LIN {X 0.323,Y -662.972,Z 876.335,A 0.000,B 0.000,C 90.000,E1 276.315} C_DIS
LIN {X 0.019,Y -659.761,Z 876.333,A 0.000,B 0.000,C 90.000,E1 275.853} C_DIS
LIN {X 0.348,Y -656.166,Z 876.330,A 0.000,B 0.000,C 90.000,E1 275.334} C_DIS
LIN {X -0.108,Y -650.680,Z 876.326,A 0.000,B 0.000,C 90.000,E1 274.759} C_DIS
LIN {X 0.134,Y -645.885,Z 876.324,A 0.000,B 0.000,C 90.000,E1 274.245} C_DIS
LIN {X -0.098,Y -638.071,Z 876.320,A 0.000,B 0.000,C 90.000,E1 273.555} C_DIS
LIN {X -0.003,Y -631.178,Z 876.317,A 0.000,B 0.000,C 90.000,E1 272.980} C_DIS
LIN {X -0.164,Y -623.612,Z 876.314,A 0.000,B 0.000,C 90.000,E1 272.465} C_DIS
LIN {X -0.009,Y -617.393,Z 876.312,A 0.000,B 0.000,C 90.000,E1 272.064} C_DIS
LIN {X -0.140,Y -610.911,Z 876.310,A 0.000,B 0.000,C 90.000,E1 271.718} C_DIS
LIN {X 0.108,Y -604.182,Z 876.308,A 0.000,B 0.000,C 90.000,E1 271.375} C_DIS
LIN {X 0.063,Y -597.337,Z 876.306,A 0.000,B 0.000,C 90.000,E1 271.088} C_DIS
LIN {X -0.214,Y -590.091,Z 876.305,A 0.000,B 0.000,C 90.000,E1 270.859} C_DIS
LIN {X -0.149,Y -584.631,Z 876.304,A 0.000,B 0.000,C 90.000,E1 270.688} C_DIS
LIN {X 0.237,Y -576.605,Z 876.303,A 0.000,B 0.000,C 90.000,E1 270.458} C_DIS
LIN {X 0.221,Y -569.921,Z 876.302,A 0.000,B 0.000,C 90.000,E1 270.344} C_DIS
LIN {X 0.254,Y -564.625,Z 876.302,A 0.000,B 0.000,C 90.000,E1 270.286} C_DIS
LIN {X 0.107,Y -553.667,Z 876.301,A 0.000,B 0.000,C 90.000,E1 270.229} C_DIS
LIN {X -0.050,Y -552.373,Z 876.301,A 0.000,B 0.000,C 90.000,E1 270.229} C_DIS
LIN {X 0.018,Y -549.331,Z 876.301,A 0.000,B 0.000,C 90.000,E1 270.115} C_DIS
LIN {X -0.108,Y -547.301,Z 876.300,A 0.000,B 0.000,C 90.000,E1 269.943} C_DIS
LIN {X -0.153,Y -546.410,Z 876.298,A 0.000,B 0.000,C 90.000,E1 269.714} C_DIS
LIN {X 0.190,Y -545.549,Z 876.296,A 0.000,B 0.000,C 90.000,E1 269.255} C_DIS
LIN {X 0.218,Y -541.822,Z 876.272,A 0.000,B 0.000,C 90.000,E1 265.008} C_DIS
LIN {X -0.161,Y -541.097,Z 876.266,A 0.000,B 0.000,C 90.000,E1 263.913} C_DIS
LIN {X 0.056,Y -540.026,Z 876.258,A 0.000,B 0.000,C 90.000,E1 262.470} C_DIS
LIN {X 0.242,Y -538.664,Z 876.250,A 0.000,B 0.000,C 90.000,E1 261.027} C_DIS
LIN {X -0.117,Y -537.550,Z 876.244,A 0.000,B 0.000,C 90.000,E1 259.926} C_DIS
LIN {X -0.273,Y -535.768,Z 876.234,A 0.000,B 0.000,C 90.000,E1 258.229} C_DIS
LIN {X -0.051,Y -534.476,Z 876.228,A 0.000,B 0.000,C 90.000,E1 257.061} C_DIS
LIN {X -0.248,Y -533.064,Z 876.222,A 0.000,B 0.000,C 90.000,E1 255.936} C_DIS
LIN {X -0.214,Y -530.574,Z 876.211,A 0.000,B 0.000,C 90.000,E1 253.921} C_DIS
LIN {X 0.057,Y -528.202,Z 876.199,A 0.000,B 0.000,C 90.000,E1 251.873} C_DIS
LIN {X -0.252,Y -527.077,Z 876.195,A 0.000,B 0.000,C 90.000,E1 251.040} C_DIS
LIN {X -0.063,Y -525.191,Z 876.187,A 0.000,B 0.000,C 90.000,E1 249.571} C_DIS
LIN {X -0.073,Y -523.643,Z 876.180,A 0.000,B 0.000,C 90.000,E1 248.411} C_DIS
LIN {X 0.243,Y -521.461,Z 876.172,A 0.000,B 0.000,C 90.000,E1 246.922} C_DIS
LIN {X -0.107,Y -519.733,Z 876.166,A 0.000,B 0.000,C 90.000,E1 245.793} C_DIS
LIN {X -0.123,Y -517.477,Z 876.157,A 0.000,B 0.000,C 90.000,E1 244.332} C_DIS
LIN {X 0.157,Y -515.575,Z 876.151,A 0.000,B 0.000,C 90.000,E1 243.127} C_DIS
LIN {X -0.056,Y -512.523,Z 876.141,A 0.000,B 0.000,C 90.000,E1 241.385} C_DIS
LIN {X -0.098,Y -509.431,Z 876.131,A 0.000,B 0.000,C 90.000,E1 239.616} C_DIS
LIN {X 0.092,Y -507.327,Z 876.125,A 0.000,B 0.000,C 90.000,E1 238.408} C_DIS
LIN {X 0.136,Y -504.494,Z 876.116,A 0.000,B 0.000,C 90.000,E1 236.914} C_DIS
LIN {X 0.107,Y -502.069,Z 876.110,A 0.000,B 0.000,C 90.000,E1 235.722} C_DIS
LIN {X 0.288,Y -500.765,Z 876.106,A 0.000,B 0.000,C 90.000,E1 235.102} C_DIS
LIN {X 0.079,Y -497.210,Z 876.098,A 0.000,B 0.000,C 90.000,E1 233.623} C_DIS
LIN {X -0.042,Y -492.982,Z 876.088,A 0.000,B 0.000,C 90.000,E1 231.823} C_DIS
LIN {X 0.202,Y -489.383,Z 876.079,A 0.000,B 0.000,C 90.000,E1 230.275} C_DIS
LIN {X -0.143,Y -486.645,Z 876.073,A 0.000,B 0.000,C 90.000,E1 229.094} C_DIS
LIN {X 0.110,Y -483.868,Z 876.066,A 0.000,B 0.000,C 90.000,E1 227.838} C_DIS
LIN {X 0.253,Y -479.873,Z 876.056,A 0.000,B 0.000,C 90.000,E1 225.972} C_DIS
LIN {X 0.285,Y -475.776,Z 876.045,A 0.000,B 0.000,C 90.000,E1 224.109} C_DIS
LIN {X -0.199,Y -472.305,Z 876.037,A 0.000,B 0.000,C 90.000,E1 222.609} C_DIS
LIN {X 0.100,Y -467.450,Z 876.024,A 0.000,B 0.000,C 90.000,E1 220.378} C_DIS
LIN {X 0.020,Y -462.719,Z 876.012,A 0.000,B 0.000,C 90.000,E1 218.177} C_DIS
LIN {X -0.203,Y -458.741,Z 876.002,A 0.000,B 0.000,C 90.000,E1 216.297} C_DIS
LIN {X 0.215,Y -454.685,Z 875.991,A 0.000,B 0.000,C 90.000,E1 214.326} C_DIS
LIN {X 0.130,Y -452.624,Z 875.986,A 0.000,B 0.000,C 90.000,E1 213.372} C_DIS
LIN {X -0.102,Y -448.540,Z 875.975,A 0.000,B 0.000,C 90.000,E1 211.465} C_DIS
LIN {X -0.219,Y -443.633,Z 875.962,A 0.000,B 0.000,C 90.000,E1 209.205} C_DIS
LIN {X 0.212,Y -440.087,Z 875.953,A 0.000,B 0.000,C 90.000,E1 207.513} C_DIS
LIN {X 0.215,Y -435.105,Z 875.940,A 0.000,B 0.000,C 90.000,E1 205.207} C_DIS
LIN {X -0.102,Y -430.943,Z 875.929,A 0.000,B 0.000,C 90.000,E1 203.259} C_DIS
LIN {X -0.085,Y -426.161,Z 875.916,A 0.000,B 0.000,C 90.000,E1 200.918} C_DIS
LIN {X 0.085,Y -422.719,Z 875.907,A 0.000,B 0.000,C 90.000,E1 199.214} C_DIS
LIN {X 0.177,Y -419.410,Z 875.897,A 0.000,B 0.000,C 90.000,E1 197.511} C_DIS
LIN {X -0.207,Y -416.674,Z 875.890,A 0.000,B 0.000,C 90.000,E1 196.205} C_DIS
LIN {X -0.081,Y -413.195,Z 875.880,A 0.000,B 0.000,C 90.000,E1 194.481} C_DIS
LIN {X 0.010,Y -408.527,Z 875.867,A 0.000,B 0.000,C 90.000,E1 192.063} C_DIS
LIN {X 0.161,Y -405.858,Z 875.859,A 0.000,B 0.000,C 90.000,E1 190.658} C_DIS
LIN {X 0.195,Y -402.402,Z 875.850,A 0.000,B 0.000,C 90.000,E1 188.916} C_DIS
LIN {X 0.064,Y -397.475,Z 875.836,A 0.000,B 0.000,C 90.000,E1 186.486} C_DIS
LIN {X 0.194,Y -390.868,Z 875.815,A 0.000,B 0.000,C 90.000,E1 182.579} C_DIS
LIN {X 0.078,Y -387.709,Z 875.803,A 0.000,B 0.000,C 90.000,E1 180.458} C_DIS
LIN {X 0.084,Y -385.689,Z 875.795,A 0.000,B 0.000,C 90.000,E1 179.026} C_DIS
LIN {X -0.046,Y -382.997,Z 875.785,A 0.000,B 0.000,C 90.000,E1 177.249} C_DIS
LIN {X -0.087,Y -380.876,Z 875.777,A 0.000,B 0.000,C 90.000,E1 175.812} C_DIS
LIN {X -0.123,Y -377.307,Z 875.763,A 0.000,B 0.000,C 90.000,E1 173.280} C_DIS
LIN {X 0.154,Y -375.585,Z 875.755,A 0.000,B 0.000,C 90.000,E1 171.781} C_DIS
LIN {X 0.082,Y -374.388,Z 875.746,A 0.000,B 0.000,C 90.000,E1 170.330} C_DIS
LIN {X 0.175,Y -373.752,Z 875.740,A 0.000,B 0.000,C 90.000,E1 169.218} C_DIS
LIN {X -0.176,Y -373.799,Z 875.734,A 0.000,B 0.000,C 90.000,E1 168.173} C_DIS
LIN {X 0.030,Y -374.075,Z 875.730,A 0.000,B 0.000,C 90.000,E1 167.409} C_DIS
LIN {X -0.125,Y -374.536,Z 875.726,A 0.000,B 0.000,C 90.000,E1 166.700} C_DIS
LIN {X 0.103,Y -375.301,Z 875.723,A 0.000,B 0.000,C 90.000,E1 166.117} C_DIS
LIN {X 0.082,Y -376.304,Z 875.721,A 0.000,B 0.000,C 90.000,E1 165.700} C_DIS
LIN {X 0.058,Y -377.044,Z 875.719,A 0.000,B 0.000,C 90.000,E1 165.338} C_DIS
LIN {X -0.058,Y -378.009,Z 875.717,A 0.000,B 0.000,C 90.000,E1 164.991} C_DIS
LIN {X 0.036,Y -379.120,Z 875.715,A 0.000,B 0.000,C 90.000,E1 164.629} C_DIS
LIN {X -0.079,Y -382.383,Z 875.712,A 0.000,B 0.000,C 90.000,E1 164.102} C_DIS
LIN {X -0.081,Y -383.396,Z 875.711,A 0.000,B 0.000,C 90.000,E1 163.921} C_DIS
LIN {X -0.077,Y -384.658,Z 875.710,A 0.000,B 0.000,C 90.000,E1 163.740} C_DIS
LIN {X 0.042,Y -390.123,Z 875.707,A 0.000,B 0.000,C 90.000,E1 163.196} C_DIS
LIN {X -0.218,Y -392.050,Z 875.706,A 0.000,B 0.000,C 90.000,E1 163.087} C_DIS
LIN {X -0.034,Y -398.644,Z 875.704,A 0.000,B 0.000,C 90.000,E1 162.670} C_DIS
LIN {X -0.002,Y -417.692,Z 875.698,A 0.000,B 0.000,C 90.000,E1 161.692} C_DIS
LIN {X 0.178,Y -422.461,Z 875.697,A 0.000,B 0.000,C 90.000,E1 161.402} C_DIS
LIN {X -0.122,Y -428.928,Z 875.695,A 0.000,B 0.000,C 90.000,E1 161.040} C_DIS
LIN {X -0.202,Y -438.322,Z 875.691,A 0.000,B 0.000,C 90.000,E1 160.369} C_DIS
LIN {X -0.136,Y -446.051,Z 875.687,A 0.000,B 0.000,C 90.000,E1 159.752} C_DIS
LIN {X -0.042,Y -456.665,Z 875.682,A 0.000,B 0.000,C 90.000,E1 158.847} C_DIS
LIN {X -0.125,Y -459.495,Z 875.681,A 0.000,B 0.000,C 90.000,E1 158.592} C_DIS
LIN {X -0.089,Y -469.554,Z 875.675,A 0.000,B 0.000,C 90.000,E1 157.592} C_DIS
LIN {X 0.090,Y -479.076,Z 875.670,A 0.000,B 0.000,C 90.000,E1 156.538} C_DIS
LIN {X -0.175,Y -489.344,Z 875.663,A 0.000,B 0.000,C 90.000,E1 155.357} C_DIS
LIN {X 0.120,Y -496.471,Z 875.658,A 0.000,B 0.000,C 90.000,E1 154.409} C_DIS
LIN {X -0.141,Y -504.231,Z 875.652,A 0.000,B 0.000,C 90.000,E1 153.384} C_DIS
LIN {X 0.054,Y -509.663,Z 875.648,A 0.000,B 0.000,C 90.000,E1 152.615} C_DIS
LIN {X 0.145,Y -519.842,Z 875.640,A 0.000,B 0.000,C 90.000,E1 151.129} C_DIS
LIN {X 0.128,Y -525.696,Z 875.635,A 0.000,B 0.000,C 90.000,E1 150.255} C_DIS
LIN {X -0.087,Y -531.123,Z 875.630,A 0.000,B 0.000,C 90.000,E1 149.410} C_DIS
LIN {X 0.024,Y -536.329,Z 875.625,A 0.000,B 0.000,C 90.000,E1 148.535} C_DIS
LIN {X -0.268,Y -539.600,Z 875.622,A 0.000,B 0.000,C 90.000,E1 147.995} C_DIS
LIN {X -0.137,Y -548.333,Z 875.613,A 0.000,B 0.000,C 90.000,E1 146.421} C_DIS
LIN {X 0.345,Y -553.510,Z 875.608,A 0.000,B 0.000,C 90.000,E1 145.388} C_DIS
LIN {X -0.216,Y -557.743,Z 875.603,A 0.000,B 0.000,C 90.000,E1 144.609} C_DIS
LIN {X -0.165,Y -561.241,Z 875.599,A 0.000,B 0.000,C 90.000,E1 143.909} C_DIS
LIN {X 0.135,Y -567.608,Z 875.593,A 0.000,B 0.000,C 90.000,E1 142.637} C_DIS
LIN {X -0.083,Y -576.334,Z 875.583,A 0.000,B 0.000,C 90.000,E1 140.884} C_DIS
LIN {X 0.091,Y -581.515,Z 875.577,A 0.000,B 0.000,C 90.000,E1 139.784} C_DIS
LIN {X 0.276,Y -586.418,Z 875.571,A 0.000,B 0.000,C 90.000,E1 138.690} C_DIS
LIN {X -0.131,Y -595.235,Z 875.560,A 0.000,B 0.000,C 90.000,E1 136.863} C_DIS
LIN {X 0.038,Y -601.513,Z 875.553,A 0.000,B 0.000,C 90.000,E1 135.526} C_DIS
LIN {X -0.276,Y -603.439,Z 875.551,A 0.000,B 0.000,C 90.000,E1 135.162} C_DIS
LIN {X 0.041,Y -609.364,Z 875.544,A 0.000,B 0.000,C 90.000,E1 133.824} C_DIS
LIN {X 0.187,Y -614.049,Z 875.538,A 0.000,B 0.000,C 90.000,E1 132.771} C_DIS
LIN {X -0.191,Y -619.680,Z 875.531,A 0.000,B 0.000,C 90.000,E1 131.515} C_DIS
LIN {X 0.128,Y -624.020,Z 875.525,A 0.000,B 0.000,C 90.000,E1 130.458} C_DIS
LIN {X 0.110,Y -628.089,Z 875.519,A 0.000,B 0.000,C 90.000,E1 129.439} C_DIS
LIN {X 0.024,Y -632.995,Z 875.512,A 0.000,B 0.000,C 90.000,E1 128.177} C_DIS
LIN {X 0.131,Y -636.916,Z 875.507,A 0.000,B 0.000,C 90.000,E1 127.156} C_DIS
LIN {X -0.093,Y -640.736,Z 875.501,A 0.000,B 0.000,C 90.000,E1 126.171} C_DIS
LIN {X 0.223,Y -643.496,Z 875.497,A 0.000,B 0.000,C 90.000,E1 125.391} C_DIS
LIN {X -0.393,Y -647.581,Z 875.490,A 0.000,B 0.000,C 90.000,E1 124.199} C_DIS
LIN {X 0.056,Y -650.606,Z 875.484,A 0.000,B 0.000,C 90.000,E1 123.166} C_DIS
LIN {X -0.356,Y -653.285,Z 875.479,A 0.000,B 0.000,C 90.000,E1 122.212} C_DIS
LIN {X -0.281,Y -655.064,Z 875.475,A 0.000,B 0.000,C 90.000,E1 121.465} C_DIS
LIN {X 0.031,Y -657.619,Z 875.468,A 0.000,B 0.000,C 90.000,E1 120.207} C_DIS
LIN {X 0.262,Y -659.283,Z 875.462,A 0.000,B 0.000,C 90.000,E1 119.205} C_DIS
LIN {X 0.063,Y -660.434,Z 875.458,A 0.000,B 0.000,C 90.000,E1 118.487} C_DIS
LIN {X 0.006,Y -661.948,Z 875.453,A 0.000,B 0.000,C 90.000,E1 117.513} C_DIS
LIN {X -0.173,Y -663.047,Z 875.449,A 0.000,B 0.000,C 90.000,E1 116.796} C_DIS
LIN {X 0.101,Y -664.310,Z 875.443,A 0.000,B 0.000,C 90.000,E1 115.796} C_DIS
LIN {X 0.082,Y -665.051,Z 875.438,A 0.000,B 0.000,C 90.000,E1 114.823} C_DIS
LIN {X 0.097,Y -665.286,Z 875.435,A 0.000,B 0.000,C 90.000,E1 114.335} C_DIS
LIN {X 0.389,Y -665.304,Z 875.433,A 0.000,B 0.000,C 90.000,E1 113.823} C_DIS
LIN {X -0.196,Y -664.753,Z 875.430,A 0.000,B 0.000,C 90.000,E1 113.387} C_DIS
LIN {X -0.054,Y -664.380,Z 875.429,A 0.000,B 0.000,C 90.000,E1 113.131} C_DIS
LIN {X 0.035,Y -661.702,Z 875.425,A 0.000,B 0.000,C 90.000,E1 112.514} C_DIS
LIN {X 0.102,Y -660.802,Z 875.424,A 0.000,B 0.000,C 90.000,E1 112.386} C_DIS
LIN {X -0.021,Y -658.470,Z 875.423,A 0.000,B 0.000,C 90.000,E1 112.153} C_DIS
LIN {X 0.044,Y -657.015,Z 875.422,A 0.000,B 0.000,C 90.000,E1 111.972} C_DIS
LIN {X 0.102,Y -655.691,Z 875.421,A 0.000,B 0.000,C 90.000,E1 111.844} C_DIS
LIN {X -0.054,Y -652.134,Z 875.420,A 0.000,B 0.000,C 90.000,E1 111.642} C_DIS
LIN {X -0.203,Y -647.809,Z 875.419,A 0.000,B 0.000,C 90.000,E1 111.408} C_DIS
LIN {X -0.086,Y -641.358,Z 875.418,A 0.000,B 0.000,C 90.000,E1 111.153} C_DIS
LIN {X 0.165,Y -630.848,Z 875.416,A 0.000,B 0.000,C 90.000,E1 110.791} C_DIS
LIN {X -0.177,Y -625.740,Z 875.415,A 0.000,B 0.000,C 90.000,E1 110.663} C_DIS
LIN {X 0.152,Y -621.263,Z 875.414,A 0.000,B 0.000,C 90.000,E1 110.482} C_DIS
LIN {X 0.066,Y -619.301,Z 875.414,A 0.000,B 0.000,C 90.000,E1 110.429} C_DIS
LIN {X -0.245,Y -610.433,Z 875.412,A 0.000,B 0.000,C 90.000,E1 110.120} C_DIS
LIN {X 0.043,Y -601.778,Z 875.410,A 0.000,B 0.000,C 90.000,E1 109.704} C_DIS
LIN {X -0.266,Y -591.984,Z 875.407,A 0.000,B 0.000,C 90.000,E1 109.268} C_DIS
LIN {X -0.114,Y -587.313,Z 875.406,A 0.000,B 0.000,C 90.000,E1 109.033} C_DIS
LIN {X -0.312,Y -578.780,Z 875.404,A 0.000,B 0.000,C 90.000,E1 108.725} C_DIS
LIN {X -0.196,Y -565.827,Z 875.402,A 0.000,B 0.000,C 90.000,E1 108.308} C_DIS
LIN {X 0.212,Y -562.764,Z 875.401,A 0.000,B 0.000,C 90.000,E1 108.127} C_DIS
LIN {X 0.156,Y -561.424,Z 875.400,A 0.000,B 0.000,C 90.000,E1 108.055} C_DIS
LIN {X -0.142,Y -559.895,Z 875.400,A 0.000,B 0.000,C 90.000,E1 107.946} C_DIS
LIN {X 0.091,Y -558.501,Z 875.398,A 0.000,B 0.000,C 90.000,E1 107.583} C_DIS
LIN {X 0.253,Y -558.033,Z 875.396,A 0.000,B 0.000,C 90.000,E1 107.221} C_DIS
LIN {X 0.017,Y -557.954,Z 875.390,A 0.000,B 0.000,C 90.000,E1 106.134} C_DIS
LIN {X 0.186,Y -559.024,Z 875.373,A 0.000,B 0.000,C 90.000,E1 103.063} C_DIS
LIN {X -0.032,Y -560.051,Z 875.363,A 0.000,B 0.000,C 90.000,E1 101.422} C_DIS
LIN {X -0.030,Y -561.573,Z 875.351,A 0.000,B 0.000,C 90.000,E1 99.208} C_DIS
LIN {X 0.167,Y -562.701,Z 875.342,A 0.000,B 0.000,C 90.000,E1 97.530} C_DIS
LIN {X 0.232,Y -563.537,Z 875.334,A 0.000,B 0.000,C 90.000,E1 96.144} C_DIS
LIN {X 0.301,Y -564.171,Z 875.327,A 0.000,B 0.000,C 90.000,E1 94.759} C_DIS
LIN {X -0.276,Y -564.766,Z 875.319,A 0.000,B 0.000,C 90.000,E1 93.440} C_DIS
LIN {X -0.271,Y -565.203,Z 875.311,A 0.000,B 0.000,C 90.000,E1 92.064} C_DIS
LIN {X -0.260,Y -565.669,Z 875.304,A 0.000,B 0.000,C 90.000,E1 90.688} C_DIS
LIN {X -0.140,Y -566.011,Z 875.295,A 0.000,B 0.000,C 90.000,E1 89.026} C_DIS
LIN {X -0.117,Y -566.258,Z 875.287,A 0.000,B 0.000,C 90.000,E1 87.650} C_DIS
LIN {X 0.171,Y -566.628,Z 875.276,A 0.000,B 0.000,C 90.000,E1 85.698} C_DIS
LIN {X -0.216,Y -566.879,Z 875.267,A 0.000,B 0.000,C 90.000,E1 84.090} C_DIS
LIN {X 0.176,Y -567.282,Z 875.256,A 0.000,B 0.000,C 90.000,E1 82.129} C_DIS
LIN {X 0.189,Y -567.890,Z 875.246,A 0.000,B 0.000,C 90.000,E1 80.208} C_DIS
LIN {X -0.146,Y -568.783,Z 875.234,A 0.000,B 0.000,C 90.000,E1 78.049} C_DIS
LIN {X 0.029,Y -569.281,Z 875.227,A 0.000,B 0.000,C 90.000,E1 76.937} C_DIS
LIN {X 0.154,Y -569.891,Z 875.218,A 0.000,B 0.000,C 90.000,E1 75.283} C_DIS
LIN {X 0.104,Y -570.360,Z 875.211,A 0.000,B 0.000,C 90.000,E1 73.921} C_DIS
LIN {X 0.042,Y -570.629,Z 875.205,A 0.000,B 0.000,C 90.000,E1 72.834} C_DIS
LIN {X -0.212,Y -570.967,Z 875.196,A 0.000,B 0.000,C 90.000,E1 71.221} C_DIS
LIN {X 0.255,Y -571.157,Z 875.185,A 0.000,B 0.000,C 90.000,E1 69.263} C_DIS
LIN {X 0.195,Y -571.268,Z 875.174,A 0.000,B 0.000,C 90.000,E1 67.358} C_DIS
LIN {X 0.162,Y -571.241,Z 875.167,A 0.000,B 0.000,C 90.000,E1 65.997} C_DIS
LIN {X -0.163,Y -571.153,Z 875.159,A 0.000,B 0.000,C 90.000,E1 64.665} C_DIS
LIN {X 0.277,Y -571.005,Z 875.152,A 0.000,B 0.000,C 90.000,E1 63.256} C_DIS
LIN {X 0.209,Y -570.687,Z 875.144,A 0.000,B 0.000,C 90.000,E1 61.897} C_DIS
LIN {X 0.238,Y -570.133,Z 875.135,A 0.000,B 0.000,C 90.000,E1 60.255} C_DIS
LIN {X 0.001,Y -569.754,Z 875.130,A 0.000,B 0.000,C 90.000,E1 59.459} C_DIS
LIN {X 0.178,Y -568.873,Z 875.123,A 0.000,B 0.000,C 90.000,E1 58.074} C_DIS
LIN {X 0.224,Y -568.272,Z 875.118,A 0.000,B 0.000,C 90.000,E1 57.248} C_DIS
LIN {X 0.267,Y -567.521,Z 875.114,A 0.000,B 0.000,C 90.000,E1 56.421} C_DIS
LIN {X 0.303,Y -566.647,Z 875.109,A 0.000,B 0.000,C 90.000,E1 55.595} C_DIS
LIN {X -0.021,Y -565.339,Z 875.103,A 0.000,B 0.000,C 90.000,E1 54.529} C_DIS
LIN {X 0.098,Y -563.814,Z 875.097,A 0.000,B 0.000,C 90.000,E1 53.417} C_DIS
LIN {X 0.077,Y -562.076,Z 875.091,A 0.000,B 0.000,C 90.000,E1 52.316} C_DIS
LIN {X 0.030,Y -560.593,Z 875.086,A 0.000,B 0.000,C 90.000,E1 51.492} C_DIS
LIN {X -0.219,Y -559.517,Z 875.083,A 0.000,B 0.000,C 90.000,E1 50.964} C_DIS
LIN {X -0.030,Y -557.698,Z 875.078,A 0.000,B 0.000,C 90.000,E1 50.114} C_DIS
LIN {X -0.214,Y -555.497,Z 875.074,A 0.000,B 0.000,C 90.000,E1 49.299} C_DIS
LIN {X -0.058,Y -553.014,Z 875.069,A 0.000,B 0.000,C 90.000,E1 48.447} C_DIS
LIN {X 0.058,Y -551.206,Z 875.066,A 0.000,B 0.000,C 90.000,E1 47.877} C_DIS
LIN {X -0.203,Y -547.058,Z 875.060,A 0.000,B 0.000,C 90.000,E1 46.782} C_DIS
LIN {X -0.165,Y -544.823,Z 875.057,A 0.000,B 0.000,C 90.000,E1 46.215} C_DIS
LIN {X -0.338,Y -543.053,Z 875.054,A 0.000,B 0.000,C 90.000,E1 45.810} C_DIS
LIN {X -0.139,Y -539.772,Z 875.050,A 0.000,B 0.000,C 90.000,E1 45.081} C_DIS
LIN {X 0.027,Y -536.128,Z 875.046,A 0.000,B 0.000,C 90.000,E1 44.352} C_DIS
LIN {X -0.191,Y -533.846,Z 875.044,A 0.000,B 0.000,C 90.000,E1 43.947} C_DIS
LIN {X 0.083,Y -528.644,Z 875.039,A 0.000,B 0.000,C 90.000,E1 43.056} C_DIS
LIN {X 0.208,Y -525.927,Z 875.037,A 0.000,B 0.000,C 90.000,E1 42.609} C_DIS
LIN {X -0.114,Y -521.051,Z 875.033,A 0.000,B 0.000,C 90.000,E1 41.919} C_DIS
LIN {X -0.025,Y -517.968,Z 875.030,A 0.000,B 0.000,C 90.000,E1 41.472} C_DIS
LIN {X -0.283,Y -511.277,Z 875.026,A 0.000,B 0.000,C 90.000,E1 40.620} C_DIS
LIN {X -0.128,Y -506.473,Z 875.022,A 0.000,B 0.000,C 90.000,E1 40.011} C_DIS
LIN {X 0.003,Y -501.274,Z 875.019,A 0.000,B 0.000,C 90.000,E1 39.402} C_DIS
LIN {X 0.104,Y -494.460,Z 875.015,A 0.000,B 0.000,C 90.000,E1 38.669} C_DIS
LIN {X 0.002,Y -490.260,Z 875.013,A 0.000,B 0.000,C 90.000,E1 38.257} C_DIS
LIN {X 0.017,Y -483.079,Z 875.009,A 0.000,B 0.000,C 90.000,E1 37.569} C_DIS
LIN {X -0.046,Y -475.646,Z 875.005,A 0.000,B 0.000,C 90.000,E1 36.916} C_DIS
LIN {X -0.017,Y -465.064,Z 875.000,A 0.000,B 0.000,C 90.000,E1 36.011} C_DIS
LIN {X -0.104,Y -452.656,Z 874.995,A 0.000,B 0.000,C 90.000,E1 35.025} C_DIS
LIN {X -0.065,Y -443.282,Z 874.990,A 0.000,B 0.000,C 90.000,E1 34.278} C_DIS
LIN {X 0.069,Y -421.693,Z 874.981,A 0.000,B 0.000,C 90.000,E1 32.498} C_DIS
LIN {X 0.024,Y -406.598,Z 874.973,A 0.000,B 0.000,C 90.000,E1 31.131} C_DIS
LIN {X -0.032,Y -399.449,Z 874.969,A 0.000,B 0.000,C 90.000,E1 30.413} C_DIS
LIN {X -0.157,Y -394.956,Z 874.966,A 0.000,B 0.000,C 90.000,E1 29.873} C_DIS
LIN {X 0.010,Y -392.401,Z 874.963,A 0.000,B 0.000,C 90.000,E1 29.411} C_DIS
LIN {X -0.057,Y -391.569,Z 874.962,A 0.000,B 0.000,C 90.000,E1 29.155} C_DIS
LIN {X 0.062,Y -390.550,Z 874.961,A 0.000,B 0.000,C 90.000,E1 28.871} C_DIS
LIN {X -0.008,Y -389.735,Z 874.958,A 0.000,B 0.000,C 90.000,E1 28.437} C_DIS
LIN {X 0.180,Y -389.516,Z 874.957,A 0.000,B 0.000,C 90.000,E1 28.231} C_DIS
LIN {X -0.109,Y -389.463,Z 874.954,A 0.000,B 0.000,C 90.000,E1 27.719} C_DIS
LIN {X 0.081,Y -389.305,Z 874.952,A 0.000,B 0.000,C 90.000,E1 27.334} C_DIS
LIN {X -0.034,Y -389.940,Z 874.944,A 0.000,B 0.000,C 90.000,E1 25.924} C_DIS
LIN {X 0.082,Y -391.522,Z 874.932,A 0.000,B 0.000,C 90.000,E1 23.770} C_DIS
LIN {X 0.169,Y -394.134,Z 874.916,A 0.000,B 0.000,C 90.000,E1 20.918} C_DIS
LIN {X -0.081,Y -396.351,Z 874.905,A 0.000,B 0.000,C 90.000,E1 18.833} C_DIS
LIN {X -0.091,Y -399.250,Z 874.891,A 0.000,B 0.000,C 90.000,E1 16.370} C_DIS
LIN {X 0.149,Y -402.374,Z 874.877,A 0.000,B 0.000,C 90.000,E1 13.883} C_DIS
LIN {X -0.094,Y -405.837,Z 874.864,A 0.000,B 0.000,C 90.000,E1 11.478} C_DIS
LIN {X 0.064,Y -410.729,Z 874.846,A 0.000,B 0.000,C 90.000,E1 8.341} C_DIS
LIN {X -0.167,Y -415.542,Z 874.831,A 0.000,B 0.000,C 90.000,E1 5.625} C_DIS
LIN {X 0.079,Y -420.777,Z 874.816,A 0.000,B 0.000,C 90.000,E1 2.865} C_DIS
LIN {X -0.204,Y -428.386,Z 874.797,A 0.000,B 0.000,C 90.000,E1 359.484} C_DIS
LIN {X 0.000,Y -434.970,Z 874.782,A 0.000,B 0.000,C 90.000,E1 356.788} C_DIS
LIN {X -0.040,Y -438.339,Z 874.775,A 0.000,B 0.000,C 90.000,E1 355.469} C_DIS
LIN {X 0.144,Y -439.863,Z 874.772,A 0.000,B 0.000,C 90.000,E1 354.951} C_DIS
LIN {X -0.037,Y -442.283,Z 874.769,A 0.000,B 0.000,C 90.000,E1 354.375} C_DIS
LIN {X 0.016,Y -443.078,Z 874.768,A 0.000,B 0.000,C 90.000,E1 354.204} C_DIS
LIN {X -0.165,Y -445.091,Z 874.766,A 0.000,B 0.000,C 90.000,E1 353.913} C_DIS
LIN {X -0.003,Y -450.120,Z 874.764,A 0.000,B 0.000,C 90.000,E1 353.451} C_DIS
LIN {X -0.228,Y -455.758,Z 874.762,A 0.000,B 0.000,C 90.000,E1 353.166} C_DIS
LIN {X 0.240,Y -470.201,Z 874.758,A 0.000,B 0.000,C 90.000,E1 352.470} C_DIS
LIN {X -0.118,Y -473.472,Z 874.758,A 0.000,B 0.000,C 90.000,E1 352.356} C_DIS
LIN {X -0.073,Y -483.315,Z 874.755,A 0.000,B 0.000,C 90.000,E1 351.837} C_DIS
LIN {X 0.204,Y -492.976,Z 874.752,A 0.000,B 0.000,C 90.000,E1 351.254} C_DIS
LIN {X -0.252,Y -504.167,Z 874.748,A 0.000,B 0.000,C 90.000,E1 350.622} C_DIS
LIN {X -0.060,Y -512.046,Z 874.745,A 0.000,B 0.000,C 90.000,E1 350.095} C_DIS
LIN {X -0.012,Y -521.344,Z 874.741,A 0.000,B 0.000,C 90.000,E1 349.454} C_DIS
LIN {X -0.201,Y -528.953,Z 874.738,A 0.000,B 0.000,C 90.000,E1 348.926} C_DIS
LIN {X -0.130,Y -534.869,Z 874.736,A 0.000,B 0.000,C 90.000,E1 348.465} C_DIS
LIN {X 0.213,Y -542.002,Z 874.733,A 0.000,B 0.000,C 90.000,E1 347.825} C_DIS
LIN {X -0.011,Y -548.932,Z 874.729,A 0.000,B 0.000,C 90.000,E1 347.229} C_DIS
LIN {X 0.203,Y -554.303,Z 874.726,A 0.000,B 0.000,C 90.000,E1 346.700} C_DIS
LIN {X 0.251,Y -559.452,Z 874.723,A 0.000,B 0.000,C 90.000,E1 346.172} C_DIS
LIN {X 0.137,Y -564.467,Z 874.720,A 0.000,B 0.000,C 90.000,E1 345.644} C_DIS
LIN {X -0.113,Y -570.323,Z 874.717,A 0.000,B 0.000,C 90.000,E1 344.991} C_DIS
LIN {X 0.146,Y -575.884,Z 874.713,A 0.000,B 0.000,C 90.000,E1 344.283} C_DIS
LIN {X -0.197,Y -582.187,Z 874.708,A 0.000,B 0.000,C 90.000,E1 343.504} C_DIS
LIN {X 0.083,Y -587.944,Z 874.704,A 0.000,B 0.000,C 90.000,E1 342.670} C_DIS
LIN {X -0.208,Y -593.976,Z 874.699,A 0.000,B 0.000,C 90.000,E1 341.764} C_DIS
LIN {X -0.126,Y -597.972,Z 874.695,A 0.000,B 0.000,C 90.000,E1 341.094} C_DIS
LIN {X -0.300,Y -603.261,Z 874.690,A 0.000,B 0.000,C 90.000,E1 340.188} C_DIS
LIN {X -0.171,Y -607.587,Z 874.685,A 0.000,B 0.000,C 90.000,E1 339.390} C_DIS
LIN {X -0.041,Y -613.104,Z 874.680,A 0.000,B 0.000,C 90.000,E1 338.337} C_DIS
LIN {X -0.067,Y -618.361,Z 874.674,A 0.000,B 0.000,C 90.000,E1 337.305} C_DIS
LIN {X -0.115,Y -623.283,Z 874.668,A 0.000,B 0.000,C 90.000,E1 336.282} C_DIS
LIN {X 0.225,Y -627.875,Z 874.663,A 0.000,B 0.000,C 90.000,E1 335.229} C_DIS
LIN {X 0.287,Y -631.062,Z 874.658,A 0.000,B 0.000,C 90.000,E1 334.460} C_DIS
LIN {X 0.184,Y -636.036,Z 874.651,A 0.000,B 0.000,C 90.000,E1 333.204} C_DIS
LIN {X -0.240,Y -638.857,Z 874.647,A 0.000,B 0.000,C 90.000,E1 332.487} C_DIS
LIN {X -0.070,Y -641.497,Z 874.643,A 0.000,B 0.000,C 90.000,E1 331.719} C_DIS
LIN {X -0.060,Y -644.822,Z 874.637,A 0.000,B 0.000,C 90.000,E1 330.717} C_DIS
LIN {X 0.090,Y -648.713,Z 874.630,A 0.000,B 0.000,C 90.000,E1 329.459} C_DIS
LIN {X 0.299,Y -652.353,Z 874.624,A 0.000,B 0.000,C 90.000,E1 328.201} C_DIS
LIN {X -0.092,Y -655.016,Z 874.618,A 0.000,B 0.000,C 90.000,E1 327.248} C_DIS
LIN {X 0.000,Y -656.913,Z 874.614,A 0.000,B 0.000,C 90.000,E1 326.501} C_DIS
LIN {X 0.129,Y -659.635,Z 874.607,A 0.000,B 0.000,C 90.000,E1 325.261} C_DIS
LIN {X -0.243,Y -661.916,Z 874.600,A 0.000,B 0.000,C 90.000,E1 324.069} C_DIS
LIN {X 0.249,Y -663.507,Z 874.595,A 0.000,B 0.000,C 90.000,E1 323.050} C_DIS
LIN {X 0.336,Y -665.221,Z 874.588,A 0.000,B 0.000,C 90.000,E1 321.823} C_DIS
LIN {X -0.009,Y -667.236,Z 874.579,A 0.000,B 0.000,C 90.000,E1 320.150} C_DIS
LIN {X 0.040,Y -668.374,Z 874.573,A 0.000,B 0.000,C 90.000,E1 319.175} C_DIS
LIN {X 0.109,Y -669.903,Z 874.565,A 0.000,B 0.000,C 90.000,E1 317.715} C_DIS
LIN {X -0.218,Y -672.654,Z 874.552,A 0.000,B 0.000,C 90.000,E1 315.324} C_DIS
LIN {X -0.156,Y -673.447,Z 874.548,A 0.000,B 0.000,C 90.000,E1 314.595} C_DIS
LIN {X 0.097,Y -675.506,Z 874.536,A 0.000,B 0.000,C 90.000,E1 312.405} C_DIS
LIN {X -0.192,Y -676.892,Z 874.528,A 0.000,B 0.000,C 90.000,E1 310.987} C_DIS
LIN {X 0.171,Y -678.488,Z 874.517,A 0.000,B 0.000,C 90.000,E1 309.036} C_DIS
LIN {X -0.040,Y -679.448,Z 874.510,A 0.000,B 0.000,C 90.000,E1 307.855} C_DIS
LIN {X -0.109,Y -680.388,Z 874.504,A 0.000,B 0.000,C 90.000,E1 306.664} C_DIS
LIN {X 0.246,Y -681.211,Z 874.497,A 0.000,B 0.000,C 90.000,E1 305.438} C_DIS
LIN {X -0.173,Y -681.965,Z 874.490,A 0.000,B 0.000,C 90.000,E1 304.278} C_DIS
LIN {X -0.003,Y -682.915,Z 874.482,A 0.000,B 0.000,C 90.000,E1 302.832} C_DIS
LIN {X -0.007,Y -684.321,Z 874.472,A 0.000,B 0.000,C 90.000,E1 300.924} C_DIS
LIN {X -0.137,Y -685.321,Z 874.465,A 0.000,B 0.000,C 90.000,E1 299.745} C_DIS
LIN {X -0.023,Y -686.635,Z 874.457,A 0.000,B 0.000,C 90.000,E1 298.309} C_DIS
LIN {X 0.341,Y -688.390,Z 874.448,A 0.000,B 0.000,C 90.000,E1 296.616} C_DIS
LIN {X 0.189,Y -689.969,Z 874.440,A 0.000,B 0.000,C 90.000,E1 295.207} C_DIS
LIN {X 0.208,Y -690.838,Z 874.435,A 0.000,B 0.000,C 90.000,E1 294.259} C_DIS
LIN {X -0.234,Y -691.135,Z 874.432,A 0.000,B 0.000,C 90.000,E1 293.823} C_DIS
LIN {X -0.040,Y -691.264,Z 874.430,A 0.000,B 0.000,C 90.000,E1 293.334} C_DIS
LIN {X 0.160,Y -690.713,Z 874.427,A 0.000,B 0.000,C 90.000,E1 292.845} C_DIS
LIN {X -0.243,Y -690.257,Z 874.426,A 0.000,B 0.000,C 90.000,E1 292.642} C_DIS
LIN {X -0.013,Y -689.271,Z 874.424,A 0.000,B 0.000,C 90.000,E1 292.386} C_DIS
LIN {X 0.065,Y -687.554,Z 874.422,A 0.000,B 0.000,C 90.000,E1 292.025} C_DIS
LIN {X 0.176,Y -686.707,Z 874.422,A 0.000,B 0.000,C 90.000,E1 291.897} C_DIS
LIN {X 0.284,Y -685.450,Z 874.421,A 0.000,B 0.000,C 90.000,E1 291.770} C_DIS
LIN {X -0.176,Y -682.244,Z 874.420,A 0.000,B 0.000,C 90.000,E1 291.589} C_DIS
LIN {X -0.321,Y -679.046,Z 874.419,A 0.000,B 0.000,C 90.000,E1 291.408} C_DIS
LIN {X 0.098,Y -677.190,Z 874.418,A 0.000,B 0.000,C 90.000,E1 291.280} C_DIS
LIN {X -0.232,Y -670.163,Z 874.417,A 0.000,B 0.000,C 90.000,E1 291.099} C_DIS
LIN {X 0.070,Y -661.113,Z 874.416,A 0.000,B 0.000,C 90.000,E1 290.844} C_DIS
LIN {X -0.092,Y -659.049,Z 874.416,A 0.000,B 0.000,C 90.000,E1 290.791} C_DIS
LIN {X 0.048,Y -653.775,Z 874.414,A 0.000,B 0.000,C 90.000,E1 290.556} C_DIS
LIN {X 0.202,Y -652.989,Z 874.414,A 0.000,B 0.000,C 90.000,E1 290.482} C_DIS
LIN {X 0.087,Y -651.522,Z 874.413,A 0.000,B 0.000,C 90.000,E1 290.355} C_DIS
LIN {X 0.045,Y -651.511,Z 874.413,A 0.000,B 0.000,C 90.000,E1 290.355} C_DIS
LIN {X 0.182,Y -651.340,Z 874.413,A 0.000,B 0.000,C 90.000,E1 290.248} C_DIS
LIN {X 0.289,Y -651.492,Z 874.412,A 0.000,B 0.000,C 90.000,E1 290.120} C_DIS
LIN {X 0.190,Y -652.461,Z 874.410,A 0.000,B 0.000,C 90.000,E1 289.758} C_DIS
LIN {X -0.131,Y -660.092,Z 874.402,A 0.000,B 0.000,C 90.000,E1 288.308} C_DIS
LIN {X -0.237,Y -663.753,Z 874.398,A 0.000,B 0.000,C 90.000,E1 287.583} C_DIS
LIN {X -0.279,Y -665.504,Z 874.396,A 0.000,B 0.000,C 90.000,E1 287.221} C_DIS
LIN {X -0.261,Y -667.585,Z 874.393,A 0.000,B 0.000,C 90.000,E1 286.732} C_DIS
LIN {X 0.145,Y -670.209,Z 874.389,A 0.000,B 0.000,C 90.000,E1 285.969} C_DIS
LIN {X 0.122,Y -672.366,Z 874.385,A 0.000,B 0.000,C 90.000,E1 285.245} C_DIS
LIN {X -0.004,Y -673.540,Z 874.382,A 0.000,B 0.000,C 90.000,E1 284.773} C_DIS
LIN {X -0.176,Y -674.883,Z 874.378,A 0.000,B 0.000,C 90.000,E1 284.064} C_DIS
LIN {X -0.283,Y -675.635,Z 874.375,A 0.000,B 0.000,C 90.000,E1 283.592} C_DIS
LIN {X 0.222,Y -676.438,Z 874.371,A 0.000,B 0.000,C 90.000,E1 282.827} C_DIS
LIN {X 0.075,Y -677.047,Z 874.367,A 0.000,B 0.000,C 90.000,E1 282.119} C_DIS
LIN {X -0.161,Y -677.224,Z 874.365,A 0.000,B 0.000,C 90.000,E1 281.658} C_DIS
LIN {X -0.257,Y -677.184,Z 874.362,A 0.000,B 0.000,C 90.000,E1 281.186} C_DIS
LIN {X 0.134,Y -676.692,Z 874.358,A 0.000,B 0.000,C 90.000,E1 280.433} C_DIS
LIN {X 0.082,Y -676.448,Z 874.357,A 0.000,B 0.000,C 90.000,E1 280.197} C_DIS
LIN {X -0.027,Y -675.711,Z 874.354,A 0.000,B 0.000,C 90.000,E1 279.726} C_DIS
LIN {X -0.256,Y -674.674,Z 874.351,A 0.000,B 0.000,C 90.000,E1 279.265} C_DIS
LIN {X 0.178,Y -673.292,Z 874.349,A 0.000,B 0.000,C 90.000,E1 278.746} C_DIS
LIN {X 0.040,Y -671.619,Z 874.346,A 0.000,B 0.000,C 90.000,E1 278.276} C_DIS
LIN {X -0.131,Y -670.719,Z 874.345,A 0.000,B 0.000,C 90.000,E1 278.049} C_DIS
LIN {X 0.281,Y -668.616,Z 874.342,A 0.000,B 0.000,C 90.000,E1 277.530} C_DIS
LIN {X 0.011,Y -665.570,Z 874.339,A 0.000,B 0.000,C 90.000,E1 276.947} C_DIS
LIN {X -0.276,Y -662.817,Z 874.336,A 0.000,B 0.000,C 90.000,E1 276.486} C_DIS
LIN {X -0.020,Y -658.783,Z 874.333,A 0.000,B 0.000,C 90.000,E1 275.853} C_DIS
LIN {X 0.304,Y -655.149,Z 874.330,A 0.000,B 0.000,C 90.000,E1 275.334} C_DIS
LIN {X -0.159,Y -649.567,Z 874.326,A 0.000,B 0.000,C 90.000,E1 274.759} C_DIS
LIN {X 0.099,Y -644.744,Z 874.324,A 0.000,B 0.000,C 90.000,E1 274.245} C_DIS
LIN {X -0.076,Y -638.228,Z 874.320,A 0.000,B 0.000,C 90.000,E1 273.669} C_DIS
LIN {X -0.004,Y -631.353,Z 874.317,A 0.000,B 0.000,C 90.000,E1 273.094} C_DIS
LIN {X -0.147,Y -623.926,Z 874.314,A 0.000,B 0.000,C 90.000,E1 272.579} C_DIS
LIN {X -0.069,Y -617.617,Z 874.312,A 0.000,B 0.000,C 90.000,E1 272.178} C_DIS
LIN {X -0.292,Y -611.022,Z 874.310,A 0.000,B 0.000,C 90.000,E1 271.833} C_DIS
LIN {X -0.151,Y -604.117,Z 874.308,A 0.000,B 0.000,C 90.000,E1 271.489} C_DIS
LIN {X -0.290,Y -597.017,Z 874.307,A 0.000,B 0.000,C 90.000,E1 271.203} C_DIS
LIN {X -0.051,Y -589.434,Z 874.305,A 0.000,B 0.000,C 90.000,E1 270.917} C_DIS
LIN {X 0.000,Y -583.938,Z 874.304,A 0.000,B 0.000,C 90.000,E1 270.745} C_DIS
LIN {X -0.231,Y -578.065,Z 874.303,A 0.000,B 0.000,C 90.000,E1 270.630} C_DIS
LIN {X -0.246,Y -571.749,Z 874.303,A 0.000,B 0.000,C 90.000,E1 270.516} C_DIS
LIN {X -0.255,Y -566.643,Z 874.302,A 0.000,B 0.000,C 90.000,E1 270.458} C_DIS
LIN {X 0.214,Y -557.376,Z 874.302,A 0.000,B 0.000,C 90.000,E1 270.344} C_DIS
LIN {X -0.064,Y -552.864,Z 874.302,A 0.000,B 0.000,C 90.000,E1 270.344} C_DIS
LIN {X 0.161,Y -549.989,Z 874.301,A 0.000,B 0.000,C 90.000,E1 270.229} C_DIS
LIN {X 0.125,Y -549.928,Z 874.301,A 0.000,B 0.000,C 90.000,E1 270.229} C_DIS
LIN {X 0.150,Y -546.961,Z 874.300,A 0.000,B 0.000,C 90.000,E1 269.943} C_DIS
LIN {X 0.110,Y -546.926,Z 874.300,A 0.000,B 0.000,C 90.000,E1 269.943} C_DIS
LIN {X -0.025,Y -546.008,Z 874.298,A 0.000,B 0.000,C 90.000,E1 269.599} C_DIS
LIN {X 0.187,Y -544.297,Z 874.290,A 0.000,B 0.000,C 90.000,E1 268.165} C_DIS
LIN {X -0.011,Y -542.117,Z 874.274,A 0.000,B 0.000,C 90.000,E1 265.355} C_DIS
LIN {X 0.215,Y -541.176,Z 874.266,A 0.000,B 0.000,C 90.000,E1 263.913} C_DIS
LIN {X -0.105,Y -540.095,Z 874.258,A 0.000,B 0.000,C 90.000,E1 262.527} C_DIS
LIN {X 0.153,Y -538.521,Z 874.249,A 0.000,B 0.000,C 90.000,E1 260.792} C_DIS
LIN {X -0.078,Y -536.786,Z 874.240,A 0.000,B 0.000,C 90.000,E1 259.106} C_DIS
LIN {X 0.105,Y -535.850,Z 874.235,A 0.000,B 0.000,C 90.000,E1 258.229} C_DIS
LIN {X -0.141,Y -534.245,Z 874.227,A 0.000,B 0.000,C 90.000,E1 256.825} C_DIS
LIN {X -0.120,Y -532.086,Z 874.217,A 0.000,B 0.000,C 90.000,E1 255.102} C_DIS
LIN {X -0.112,Y -529.671,Z 874.206,A 0.000,B 0.000,C 90.000,E1 253.087} C_DIS
LIN {X -0.052,Y -528.000,Z 874.198,A 0.000,B 0.000,C 90.000,E1 251.638} C_DIS
LIN {X 0.148,Y -525.725,Z 874.188,A 0.000,B 0.000,C 90.000,E1 249.880} C_DIS
LIN {X -0.177,Y -523.758,Z 874.180,A 0.000,B 0.000,C 90.000,E1 248.465} C_DIS
LIN {X 0.302,Y -521.155,Z 874.171,A 0.000,B 0.000,C 90.000,E1 246.666} C_DIS
LIN {X -0.050,Y -519.399,Z 874.164,A 0.000,B 0.000,C 90.000,E1 245.537} C_DIS
LIN {X -0.070,Y -517.145,Z 874.156,A 0.000,B 0.000,C 90.000,E1 244.076} C_DIS
LIN {X 0.204,Y -515.217,Z 874.149,A 0.000,B 0.000,C 90.000,E1 242.871} C_DIS
LIN {X -0.020,Y -512.144,Z 874.140,A 0.000,B 0.000,C 90.000,E1 241.129} C_DIS
LIN {X -0.048,Y -510.080,Z 874.133,A 0.000,B 0.000,C 90.000,E1 239.950} C_DIS
LIN {X 0.046,Y -507.446,Z 874.125,A 0.000,B 0.000,C 90.000,E1 238.456} C_DIS
LIN {X -0.284,Y -504.035,Z 874.115,A 0.000,B 0.000,C 90.000,E1 236.707} C_DIS
LIN {X 0.095,Y -501.586,Z 874.108,A 0.000,B 0.000,C 90.000,E1 235.468} C_DIS
LIN {X -0.102,Y -498.061,Z 874.100,A 0.000,B 0.000,C 90.000,E1 233.989} C_DIS
LIN {X -0.067,Y -494.460,Z 874.092,A 0.000,B 0.000,C 90.000,E1 232.477} C_DIS
LIN {X 0.199,Y -492.344,Z 874.086,A 0.000,B 0.000,C 90.000,E1 231.537} C_DIS
LIN {X -0.101,Y -489.488,Z 874.080,A 0.000,B 0.000,C 90.000,E1 230.356} C_DIS
LIN {X -0.126,Y -486.753,Z 874.073,A 0.000,B 0.000,C 90.000,E1 229.138} C_DIS
LIN {X -0.048,Y -483.278,Z 874.064,A 0.000,B 0.000,C 90.000,E1 227.595} C_DIS
LIN {X -0.042,Y -479.970,Z 874.056,A 0.000,B 0.000,C 90.000,E1 226.053} C_DIS
LIN {X -0.004,Y -475.938,Z 874.046,A 0.000,B 0.000,C 90.000,E1 224.190} C_DIS
LIN {X -0.041,Y -471.714,Z 874.035,A 0.000,B 0.000,C 90.000,E1 222.324} C_DIS
LIN {X 0.247,Y -466.935,Z 874.023,A 0.000,B 0.000,C 90.000,E1 220.092} C_DIS
LIN {X 0.156,Y -462.199,Z 874.011,A 0.000,B 0.000,C 90.000,E1 217.890} C_DIS
LIN {X -0.080,Y -458.194,Z 874.000,A 0.000,B 0.000,C 90.000,E1 216.011} C_DIS
LIN {X 0.067,Y -454.165,Z 873.989,A 0.000,B 0.000,C 90.000,E1 214.072} C_DIS
LIN {X -0.102,Y -448.697,Z 873.975,A 0.000,B 0.000,C 90.000,E1 211.514} C_DIS
LIN {X 0.103,Y -444.432,Z 873.964,A 0.000,B 0.000,C 90.000,E1 209.539} C_DIS
LIN {X 0.162,Y -440.983,Z 873.955,A 0.000,B 0.000,C 90.000,E1 207.897} C_DIS
LIN {X 0.189,Y -435.997,Z 873.942,A 0.000,B 0.000,C 90.000,E1 205.591} C_DIS
LIN {X 0.113,Y -431.146,Z 873.930,A 0.000,B 0.000,C 90.000,E1 203.281} C_DIS
LIN {X 0.102,Y -427.058,Z 873.918,A 0.000,B 0.000,C 90.000,E1 201.280} C_DIS
LIN {X 0.073,Y -422.927,Z 873.907,A 0.000,B 0.000,C 90.000,E1 199.268} C_DIS
LIN {X 0.040,Y -419.644,Z 873.898,A 0.000,B 0.000,C 90.000,E1 197.583} C_DIS
LIN {X 0.183,Y -416.935,Z 873.890,A 0.000,B 0.000,C 90.000,E1 196.205} C_DIS
LIN {X -0.089,Y -413.446,Z 873.881,A 0.000,B 0.000,C 90.000,E1 194.537} C_DIS
LIN {X 0.004,Y -408.754,Z 873.867,A 0.000,B 0.000,C 90.000,E1 192.119} C_DIS
LIN {X 0.169,Y -405.407,Z 873.858,A 0.000,B 0.000,C 90.000,E1 190.366} C_DIS
LIN {X 0.194,Y -402.669,Z 873.850,A 0.000,B 0.000,C 90.000,E1 188.973} C_DIS
LIN {X 0.087,Y -398.417,Z 873.838,A 0.000,B 0.000,C 90.000,E1 186.891} C_DIS
LIN {X -0.185,Y -391.092,Z 873.815,A 0.000,B 0.000,C 90.000,E1 182.694} C_DIS
LIN {X 0.185,Y -388.459,Z 873.805,A 0.000,B 0.000,C 90.000,E1 180.859} C_DIS
LIN {X 0.104,Y -385.931,Z 873.795,A 0.000,B 0.000,C 90.000,E1 179.083} C_DIS
LIN {X -0.022,Y -383.261,Z 873.785,A 0.000,B 0.000,C 90.000,E1 177.306} C_DIS
LIN {X -0.057,Y -381.136,Z 873.777,A 0.000,B 0.000,C 90.000,E1 175.869} C_DIS
LIN {X 0.016,Y -378.098,Z 873.765,A 0.000,B 0.000,C 90.000,E1 173.685} C_DIS
LIN {X -0.173,Y -375.766,Z 873.755,A 0.000,B 0.000,C 90.000,E1 171.894} C_DIS
LIN {X 0.157,Y -373.704,Z 873.741,A 0.000,B 0.000,C 90.000,E1 169.285} C_DIS
LIN {X -0.124,Y -373.590,Z 873.735,A 0.000,B 0.000,C 90.000,E1 168.229} C_DIS
LIN {X 0.080,Y -373.736,Z 873.730,A 0.000,B 0.000,C 90.000,E1 167.465} C_DIS
LIN {X -0.040,Y -373.981,Z 873.728,A 0.000,B 0.000,C 90.000,E1 167.117} C_DIS
LIN {X -0.077,Y -374.048,Z 873.726,A 0.000,B 0.000,C 90.000,E1 166.756} C_DIS
LIN {X 0.029,Y -374.970,Z 873.721,A 0.000,B 0.000,C 90.000,E1 165.825} C_DIS
LIN {X -0.134,Y -376.669,Z 873.716,A 0.000,B 0.000,C 90.000,E1 164.936} C_DIS
LIN {X -0.139,Y -378.189,Z 873.713,A 0.000,B 0.000,C 90.000,E1 164.393} C_DIS
LIN {X 0.213,Y -379.832,Z 873.711,A 0.000,B 0.000,C 90.000,E1 163.976} C_DIS
LIN {X 0.208,Y -380.846,Z 873.710,A 0.000,B 0.000,C 90.000,E1 163.795} C_DIS
LIN {X 0.106,Y -385.962,Z 873.706,A 0.000,B 0.000,C 90.000,E1 163.087} C_DIS
LIN {X 0.086,Y -391.548,Z 873.703,A 0.000,B 0.000,C 90.000,E1 162.598} C_DIS
LIN {X -0.192,Y -396.057,Z 873.702,A 0.000,B 0.000,C 90.000,E1 162.362} C_DIS
LIN {X -0.012,Y -401.350,Z 873.700,A 0.000,B 0.000,C 90.000,E1 162.054} C_DIS
LIN {X 0.003,Y -410.030,Z 873.698,A 0.000,B 0.000,C 90.000,E1 161.638} C_DIS
LIN {X 0.171,Y -420.219,Z 873.695,A 0.000,B 0.000,C 90.000,E1 161.094} C_DIS
LIN {X -0.150,Y -429.805,Z 873.692,A 0.000,B 0.000,C 90.000,E1 160.550} C_DIS
LIN {X -0.009,Y -440.598,Z 873.688,A 0.000,B 0.000,C 90.000,E1 159.752} C_DIS
LIN {X -0.026,Y -448.291,Z 873.684,A 0.000,B 0.000,C 90.000,E1 159.156} C_DIS
LIN {X -0.197,Y -455.894,Z 873.681,A 0.000,B 0.000,C 90.000,E1 158.539} C_DIS
LIN {X 0.062,Y -465.899,Z 873.675,A 0.000,B 0.000,C 90.000,E1 157.539} C_DIS
LIN {X -0.147,Y -476.925,Z 873.669,A 0.000,B 0.000,C 90.000,E1 156.410} C_DIS
LIN {X -0.227,Y -485.993,Z 873.663,A 0.000,B 0.000,C 90.000,E1 155.357} C_DIS
LIN {X 0.002,Y -491.078,Z 873.660,A 0.000,B 0.000,C 90.000,E1 154.717} C_DIS
LIN {X 0.230,Y -499.087,Z 873.654,A 0.000,B 0.000,C 90.000,E1 153.640} C_DIS
LIN {X -0.169,Y -507.954,Z 873.647,A 0.000,B 0.000,C 90.000,E1 152.487} C_DIS
LIN {X -0.225,Y -516.143,Z 873.641,A 0.000,B 0.000,C 90.000,E1 151.307} C_DIS
LIN {X -0.205,Y -520.199,Z 873.637,A 0.000,B 0.000,C 90.000,E1 150.717} C_DIS
LIN {X -0.155,Y -524.177,Z 873.634,A 0.000,B 0.000,C 90.000,E1 150.127} C_DIS
LIN {X 0.026,Y -531.384,Z 873.628,A 0.000,B 0.000,C 90.000,E1 148.948} C_DIS
LIN {X 0.140,Y -536.516,Z 873.623,A 0.000,B 0.000,C 90.000,E1 148.074} C_DIS
LIN {X -0.268,Y -543.782,Z 873.616,A 0.000,B 0.000,C 90.000,E1 146.834} C_DIS
LIN {X 0.110,Y -547.703,Z 873.612,A 0.000,B 0.000,C 90.000,E1 146.087} C_DIS
LIN {X 0.130,Y -552.854,Z 873.606,A 0.000,B 0.000,C 90.000,E1 145.102} C_DIS
LIN {X -0.058,Y -555.778,Z 873.603,A 0.000,B 0.000,C 90.000,E1 144.562} C_DIS
LIN {X -0.029,Y -559.242,Z 873.599,A 0.000,B 0.000,C 90.000,E1 143.863} C_DIS
LIN {X -0.202,Y -563.551,Z 873.595,A 0.000,B 0.000,C 90.000,E1 143.050} C_DIS
LIN {X 0.011,Y -568.387,Z 873.589,A 0.000,B 0.000,C 90.000,E1 142.065} C_DIS
LIN {X -0.231,Y -575.233,Z 873.582,A 0.000,B 0.000,C 90.000,E1 140.723} C_DIS
LIN {X -0.228,Y -579.192,Z 873.577,A 0.000,B 0.000,C 90.000,E1 139.908} C_DIS
LIN {X 0.367,Y -584.189,Z 873.571,A 0.000,B 0.000,C 90.000,E1 138.771} C_DIS
LIN {X 0.206,Y -593.700,Z 873.560,A 0.000,B 0.000,C 90.000,E1 136.782} C_DIS
LIN {X 0.363,Y -597.541,Z 873.556,A 0.000,B 0.000,C 90.000,E1 135.972} C_DIS
LIN {X -0.070,Y -602.559,Z 873.550,A 0.000,B 0.000,C 90.000,E1 134.960} C_DIS
LIN {X 0.036,Y -609.770,Z 873.541,A 0.000,B 0.000,C 90.000,E1 133.380} C_DIS
LIN {X -0.126,Y -616.597,Z 873.532,A 0.000,B 0.000,C 90.000,E1 131.838} C_DIS
LIN {X -0.001,Y -622.097,Z 873.525,A 0.000,B 0.000,C 90.000,E1 130.539} C_DIS
LIN {X -0.045,Y -626.198,Z 873.520,A 0.000,B 0.000,C 90.000,E1 129.519} C_DIS
LIN {X -0.161,Y -631.088,Z 873.513,A 0.000,B 0.000,C 90.000,E1 128.257} C_DIS
LIN {X 0.298,Y -635.949,Z 873.505,A 0.000,B 0.000,C 90.000,E1 126.950} C_DIS
LIN {X 0.067,Y -639.745,Z 873.500,A 0.000,B 0.000,C 90.000,E1 125.964} C_DIS
LIN {X -0.152,Y -642.388,Z 873.496,A 0.000,B 0.000,C 90.000,E1 125.231} C_DIS
LIN {X 0.223,Y -645.697,Z 873.490,A 0.000,B 0.000,C 90.000,E1 124.199} C_DIS
LIN {X 0.105,Y -648.750,Z 873.485,A 0.000,B 0.000,C 90.000,E1 123.214} C_DIS
LIN {X 0.215,Y -651.374,Z 873.479,A 0.000,B 0.000,C 90.000,E1 122.212} C_DIS
LIN {X 0.273,Y -653.136,Z 873.475,A 0.000,B 0.000,C 90.000,E1 121.465} C_DIS
LIN {X 0.009,Y -654.739,Z 873.471,A 0.000,B 0.000,C 90.000,E1 120.747} C_DIS
LIN {X 0.096,Y -656.145,Z 873.467,A 0.000,B 0.000,C 90.000,E1 120.001} C_DIS
LIN {X -0.014,Y -657.835,Z 873.461,A 0.000,B 0.000,C 90.000,E1 119.027} C_DIS
LIN {X 0.009,Y -660.461,Z 873.452,A 0.000,B 0.000,C 90.000,E1 117.308} C_DIS
LIN {X -0.350,Y -661.908,Z 873.446,A 0.000,B 0.000,C 90.000,E1 116.360} C_DIS
LIN {X 0.062,Y -662.752,Z 873.442,A 0.000,B 0.000,C 90.000,E1 115.591} C_DIS
LIN {X -0.122,Y -663.565,Z 873.435,A 0.000,B 0.000,C 90.000,E1 114.387} C_DIS
LIN {X -0.113,Y -663.625,Z 873.433,A 0.000,B 0.000,C 90.000,E1 113.898} C_DIS
LIN {X 0.167,Y -663.054,Z 873.430,A 0.000,B 0.000,C 90.000,E1 113.387} C_DIS
LIN {X 0.044,Y -662.621,Z 873.429,A 0.000,B 0.000,C 90.000,E1 113.153} C_DIS
LIN {X 0.313,Y -660.665,Z 873.426,A 0.000,B 0.000,C 90.000,E1 112.642} C_DIS
LIN {X 0.377,Y -660.075,Z 873.425,A 0.000,B 0.000,C 90.000,E1 112.514} C_DIS
LIN {X -0.239,Y -656.041,Z 873.423,A 0.000,B 0.000,C 90.000,E1 112.078} C_DIS
LIN {X -0.182,Y -654.857,Z 873.422,A 0.000,B 0.000,C 90.000,E1 111.950} C_DIS
LIN {X -0.308,Y -647.907,Z 873.420,A 0.000,B 0.000,C 90.000,E1 111.535} C_DIS
LIN {X 0.095,Y -646.050,Z 873.419,A 0.000,B 0.000,C 90.000,E1 111.408} C_DIS
LIN {X -0.312,Y -639.969,Z 873.418,A 0.000,B 0.000,C 90.000,E1 111.227} C_DIS
LIN {X -0.171,Y -637.218,Z 873.417,A 0.000,B 0.000,C 90.000,E1 111.099} C_DIS
LIN {X -0.035,Y -633.800,Z 873.417,A 0.000,B 0.000,C 90.000,E1 110.972} C_DIS
LIN {X -0.082,Y -630.940,Z 873.416,A 0.000,B 0.000,C 90.000,E1 110.865} C_DIS
LIN {X -0.129,Y -626.740,Z 873.415,A 0.000,B 0.000,C 90.000,E1 110.737} C_DIS
LIN {X -0.148,Y -621.218,Z 873.414,A 0.000,B 0.000,C 90.000,E1 110.536} C_DIS
LIN {X -0.333,Y -617.609,Z 873.413,A 0.000,B 0.000,C 90.000,E1 110.429} C_DIS
LIN {X -0.247,Y -608.812,Z 873.411,A 0.000,B 0.000,C 90.000,E1 110.066} C_DIS
LIN {X -0.181,Y -594.622,Z 873.408,A 0.000,B 0.000,C 90.000,E1 109.396} C_DIS
LIN {X 0.045,Y -589.583,Z 873.406,A 0.000,B 0.000,C 90.000,E1 109.141} C_DIS
LIN {X -0.297,Y -586.279,Z 873.406,A 0.000,B 0.000,C 90.000,E1 109.033} C_DIS
LIN {X 0.085,Y -579.050,Z 873.404,A 0.000,B 0.000,C 90.000,E1 108.725} C_DIS
LIN {X -0.234,Y -566.287,Z 873.402,A 0.000,B 0.000,C 90.000,E1 108.362} C_DIS
LIN {X 0.058,Y -561.884,Z 873.401,A 0.000,B 0.000,C 90.000,E1 108.127} C_DIS
LIN {X 0.113,Y -560.040,Z 873.400,A 0.000,B 0.000,C 90.000,E1 107.946} C_DIS
LIN {X 0.233,Y -558.775,Z 873.398,A 0.000,B 0.000,C 90.000,E1 107.638} C_DIS
LIN {X 0.154,Y -558.161,Z 873.395,A 0.000,B 0.000,C 90.000,E1 107.094} C_DIS
LIN {X 0.179,Y -559.279,Z 873.372,A 0.000,B 0.000,C 90.000,E1 102.939} C_DIS
LIN {X 0.105,Y -560.466,Z 873.361,A 0.000,B 0.000,C 90.000,E1 101.007} C_DIS
LIN {X -0.198,Y -561.658,Z 873.352,A 0.000,B 0.000,C 90.000,E1 99.378} C_DIS
LIN {X -0.008,Y -562.774,Z 873.343,A 0.000,B 0.000,C 90.000,E1 97.701} C_DIS
LIN {X 0.053,Y -563.656,Z 873.335,A 0.000,B 0.000,C 90.000,E1 96.315} C_DIS
LIN {X 0.073,Y -564.269,Z 873.328,A 0.000,B 0.000,C 90.000,E1 94.935} C_DIS
LIN {X 0.105,Y -564.874,Z 873.320,A 0.000,B 0.000,C 90.000,E1 93.555} C_DIS
LIN {X 0.113,Y -565.324,Z 873.312,A 0.000,B 0.000,C 90.000,E1 92.178} C_DIS
LIN {X 0.125,Y -565.791,Z 873.305,A 0.000,B 0.000,C 90.000,E1 90.802} C_DIS
LIN {X 0.248,Y -566.141,Z 873.295,A 0.000,B 0.000,C 90.000,E1 89.141} C_DIS
LIN {X 0.274,Y -566.392,Z 873.288,A 0.000,B 0.000,C 90.000,E1 87.764} C_DIS
LIN {X 0.003,Y -566.754,Z 873.277,A 0.000,B 0.000,C 90.000,E1 85.869} C_DIS
LIN {X 0.081,Y -566.959,Z 873.269,A 0.000,B 0.000,C 90.000,E1 84.489} C_DIS
LIN {X -0.144,Y -567.354,Z 873.259,A 0.000,B 0.000,C 90.000,E1 82.591} C_DIS
LIN {X 0.252,Y -567.802,Z 873.250,A 0.000,B 0.000,C 90.000,E1 80.905} C_DIS
LIN {X 0.185,Y -568.509,Z 873.239,A 0.000,B 0.000,C 90.000,E1 78.993} C_DIS
LIN {X -0.216,Y -569.408,Z 873.228,A 0.000,B 0.000,C 90.000,E1 77.117} C_DIS
LIN {X 0.087,Y -570.064,Z 873.218,A 0.000,B 0.000,C 90.000,E1 75.172} C_DIS
LIN {X -0.179,Y -570.601,Z 873.209,A 0.000,B 0.000,C 90.000,E1 73.559} C_DIS
LIN {X 0.312,Y -570.808,Z 873.203,A 0.000,B 0.000,C 90.000,E1 72.417} C_DIS
LIN {X 0.081,Y -571.055,Z 873.196,A 0.000,B 0.000,C 90.000,E1 71.348} C_DIS
LIN {X 0.161,Y -571.253,Z 873.184,A 0.000,B 0.000,C 90.000,E1 69.156} C_DIS
LIN {X 0.310,Y -571.325,Z 873.174,A 0.000,B 0.000,C 90.000,E1 67.230} C_DIS
LIN {X -0.242,Y -571.285,Z 873.166,A 0.000,B 0.000,C 90.000,E1 65.921} C_DIS
LIN {X -0.044,Y -571.151,Z 873.159,A 0.000,B 0.000,C 90.000,E1 64.537} C_DIS
LIN {X -0.112,Y -570.978,Z 873.151,A 0.000,B 0.000,C 90.000,E1 63.179} C_DIS
LIN {X 0.328,Y -570.626,Z 873.143,A 0.000,B 0.000,C 90.000,E1 61.769} C_DIS
LIN {X -0.250,Y -570.170,Z 873.136,A 0.000,B 0.000,C 90.000,E1 60.461} C_DIS
LIN {X 0.005,Y -569.814,Z 873.131,A 0.000,B 0.000,C 90.000,E1 59.616} C_DIS
LIN {X -0.195,Y -568.712,Z 873.122,A 0.000,B 0.000,C 90.000,E1 57.995} C_DIS
LIN {X -0.148,Y -568.086,Z 873.118,A 0.000,B 0.000,C 90.000,E1 57.168} C_DIS
LIN {X -0.221,Y -567.603,Z 873.115,A 0.000,B 0.000,C 90.000,E1 56.628} C_DIS
LIN {X -0.067,Y -566.367,Z 873.108,A 0.000,B 0.000,C 90.000,E1 55.515} C_DIS
LIN {X 0.070,Y -565.032,Z 873.102,A 0.000,B 0.000,C 90.000,E1 54.402} C_DIS
LIN {X 0.178,Y -563.450,Z 873.096,A 0.000,B 0.000,C 90.000,E1 53.290} C_DIS
LIN {X 0.148,Y -561.655,Z 873.090,A 0.000,B 0.000,C 90.000,E1 52.190} C_DIS
LIN {X 0.004,Y -560.114,Z 873.085,A 0.000,B 0.000,C 90.000,E1 51.376} C_DIS
LIN {X -0.153,Y -558.348,Z 873.081,A 0.000,B 0.000,C 90.000,E1 50.561} C_DIS
LIN {X 0.017,Y -557.054,Z 873.078,A 0.000,B 0.000,C 90.000,E1 49.989} C_DIS
LIN {X -0.179,Y -554.787,Z 873.073,A 0.000,B 0.000,C 90.000,E1 49.175} C_DIS
LIN {X -0.096,Y -553.178,Z 873.070,A 0.000,B 0.000,C 90.000,E1 48.609} C_DIS
LIN {X 0.035,Y -550.337,Z 873.065,A 0.000,B 0.000,C 90.000,E1 47.757} C_DIS
LIN {X 0.135,Y -547.176,Z 873.061,A 0.000,B 0.000,C 90.000,E1 46.905} C_DIS
LIN {X -0.201,Y -544.985,Z 873.058,A 0.000,B 0.000,C 90.000,E1 46.377} C_DIS
LIN {X -0.177,Y -542.607,Z 873.054,A 0.000,B 0.000,C 90.000,E1 45.810} C_DIS
LIN {X 0.018,Y -539.246,Z 873.051,A 0.000,B 0.000,C 90.000,E1 45.081} C_DIS
LIN {X 0.180,Y -535.546,Z 873.047,A 0.000,B 0.000,C 90.000,E1 44.352} C_DIS
LIN {X -0.043,Y -533.230,Z 873.044,A 0.000,B 0.000,C 90.000,E1 43.947} C_DIS
LIN {X 0.058,Y -528.849,Z 873.040,A 0.000,B 0.000,C 90.000,E1 43.218} C_DIS
LIN {X 0.344,Y -525.183,Z 873.037,A 0.000,B 0.000,C 90.000,E1 42.609} C_DIS
LIN {X -0.135,Y -521.244,Z 873.034,A 0.000,B 0.000,C 90.000,E1 42.081} C_DIS
LIN {X -0.044,Y -518.216,Z 873.031,A 0.000,B 0.000,C 90.000,E1 41.634} C_DIS
LIN {X 0.035,Y -511.497,Z 873.026,A 0.000,B 0.000,C 90.000,E1 40.744} C_DIS
LIN {X -0.024,Y -505.416,Z 873.022,A 0.000,B 0.000,C 90.000,E1 40.011} C_DIS
LIN {X -0.062,Y -500.279,Z 873.019,A 0.000,B 0.000,C 90.000,E1 39.439} C_DIS
LIN {X 0.080,Y -493.447,Z 873.015,A 0.000,B 0.000,C 90.000,E1 38.705} C_DIS
LIN {X -0.195,Y -487.767,Z 873.012,A 0.000,B 0.000,C 90.000,E1 38.177} C_DIS
LIN {X -0.259,Y -480.660,Z 873.008,A 0.000,B 0.000,C 90.000,E1 37.523} C_DIS
LIN {X -0.012,Y -471.598,Z 873.004,A 0.000,B 0.000,C 90.000,E1 36.710} C_DIS
LIN {X 0.072,Y -462.751,Z 873.000,A 0.000,B 0.000,C 90.000,E1 35.964} C_DIS
LIN {X 0.056,Y -450.407,Z 872.994,A 0.000,B 0.000,C 90.000,E1 34.978} C_DIS
LIN {X -0.140,Y -434.922,Z 872.988,A 0.000,B 0.000,C 90.000,E1 33.785} C_DIS
LIN {X -0.033,Y -413.606,Z 872.978,A 0.000,B 0.000,C 90.000,E1 31.957} C_DIS
LIN {X -0.168,Y -404.641,Z 872.973,A 0.000,B 0.000,C 90.000,E1 31.131} C_DIS
LIN {X 0.110,Y -398.057,Z 872.969,A 0.000,B 0.000,C 90.000,E1 30.384} C_DIS
LIN {X 0.184,Y -394.244,Z 872.966,A 0.000,B 0.000,C 90.000,E1 29.873} C_DIS
LIN {X -0.138,Y -392.741,Z 872.965,A 0.000,B 0.000,C 90.000,E1 29.667} C_DIS
LIN {X 0.073,Y -392.021,Z 872.964,A 0.000,B 0.000,C 90.000,E1 29.489} C_DIS
LIN {X 0.105,Y -390.127,Z 872.960,A 0.000,B 0.000,C 90.000,E1 28.821} C_DIS
LIN {X 0.014,Y -389.475,Z 872.957,A 0.000,B 0.000,C 90.000,E1 28.309} C_DIS
LIN {X -0.081,Y -389.430,Z 872.951,A 0.000,B 0.000,C 90.000,E1 27.257} C_DIS
LIN {X -0.009,Y -390.398,Z 872.942,A 0.000,B 0.000,C 90.000,E1 25.463} C_DIS
LIN {X -0.086,Y -391.760,Z 872.932,A 0.000,B 0.000,C 90.000,E1 23.695} C_DIS
LIN {X -0.001,Y -394.395,Z 872.916,A 0.000,B 0.000,C 90.000,E1 20.844} C_DIS
LIN {X -0.074,Y -396.246,Z 872.906,A 0.000,B 0.000,C 90.000,E1 19.087} C_DIS
LIN {X 0.001,Y -399.509,Z 872.890,A 0.000,B 0.000,C 90.000,E1 16.260} C_DIS
LIN {X -0.133,Y -402.626,Z 872.877,A 0.000,B 0.000,C 90.000,E1 13.828} C_DIS
LIN {X 0.025,Y -405.618,Z 872.865,A 0.000,B 0.000,C 90.000,E1 11.715} C_DIS
LIN {X -0.187,Y -409.893,Z 872.850,A 0.000,B 0.000,C 90.000,E1 8.973} C_DIS
LIN {X -0.006,Y -415.231,Z 872.833,A 0.000,B 0.000,C 90.000,E1 5.853} C_DIS
LIN {X -0.193,Y -420.424,Z 872.817,A 0.000,B 0.000,C 90.000,E1 3.151} C_DIS
LIN {X -0.202,Y -428.526,Z 872.797,A 0.000,B 0.000,C 90.000,E1 359.484} C_DIS
LIN {X 0.004,Y -435.098,Z 872.782,A 0.000,B 0.000,C 90.000,E1 356.788} C_DIS
LIN {X 0.101,Y -439.364,Z 872.773,A 0.000,B 0.000,C 90.000,E1 355.122} C_DIS
LIN {X -0.093,Y -441.660,Z 872.769,A 0.000,B 0.000,C 90.000,E1 354.489} C_DIS
LIN {X 0.117,Y -444.026,Z 872.767,A 0.000,B 0.000,C 90.000,E1 353.970} C_DIS
LIN {X 0.174,Y -445.149,Z 872.766,A 0.000,B 0.000,C 90.000,E1 353.799} C_DIS
LIN {X -0.075,Y -449.779,Z 872.763,A 0.000,B 0.000,C 90.000,E1 353.394} C_DIS
LIN {X 0.155,Y -456.061,Z 872.761,A 0.000,B 0.000,C 90.000,E1 352.996} C_DIS
LIN {X -0.183,Y -468.866,Z 872.758,A 0.000,B 0.000,C 90.000,E1 352.470} C_DIS
LIN {X 0.121,Y -478.434,Z 872.755,A 0.000,B 0.000,C 90.000,E1 351.951} C_DIS
LIN {X -0.064,Y -486.393,Z 872.753,A 0.000,B 0.000,C 90.000,E1 351.546} C_DIS
LIN {X -0.141,Y -494.464,Z 872.750,A 0.000,B 0.000,C 90.000,E1 351.084} C_DIS
LIN {X 0.191,Y -502.345,Z 872.748,A 0.000,B 0.000,C 90.000,E1 350.566} C_DIS
LIN {X -0.057,Y -511.809,Z 872.744,A 0.000,B 0.000,C 90.000,E1 349.982} C_DIS
LIN {X -0.017,Y -519.536,Z 872.741,A 0.000,B 0.000,C 90.000,E1 349.454} C_DIS
LIN {X -0.195,Y -527.206,Z 872.738,A 0.000,B 0.000,C 90.000,E1 348.926} C_DIS
LIN {X -0.069,Y -533.200,Z 872.736,A 0.000,B 0.000,C 90.000,E1 348.465} C_DIS
LIN {X -0.148,Y -543.095,Z 872.731,A 0.000,B 0.000,C 90.000,E1 347.645} C_DIS
LIN {X 0.129,Y -550.019,Z 872.728,A 0.000,B 0.000,C 90.000,E1 346.992} C_DIS
LIN {X 0.303,Y -555.312,Z 872.725,A 0.000,B 0.000,C 90.000,E1 346.464} C_DIS
LIN {X -0.210,Y -560.461,Z 872.722,A 0.000,B 0.000,C 90.000,E1 345.992} C_DIS
LIN {X 0.244,Y -565.403,Z 872.719,A 0.000,B 0.000,C 90.000,E1 345.408} C_DIS
LIN {X -0.008,Y -571.263,Z 872.715,A 0.000,B 0.000,C 90.000,E1 344.755} C_DIS
LIN {X 0.062,Y -578.944,Z 872.710,A 0.000,B 0.000,C 90.000,E1 343.795} C_DIS
LIN {X -0.162,Y -584.023,Z 872.706,A 0.000,B 0.000,C 90.000,E1 343.142} C_DIS
LIN {X -0.170,Y -588.724,Z 872.703,A 0.000,B 0.000,C 90.000,E1 342.472} C_DIS
LIN {X 0.120,Y -594.737,Z 872.697,A 0.000,B 0.000,C 90.000,E1 341.511} C_DIS
LIN {X -0.084,Y -600.228,Z 872.692,A 0.000,B 0.000,C 90.000,E1 340.604} C_DIS
LIN {X 0.264,Y -606.881,Z 872.686,A 0.000,B 0.000,C 90.000,E1 339.390} C_DIS
LIN {X 0.119,Y -613.773,Z 872.678,A 0.000,B 0.000,C 90.000,E1 338.103} C_DIS
LIN {X -0.235,Y -619.016,Z 872.673,A 0.000,B 0.000,C 90.000,E1 337.102} C_DIS
LIN {X 0.052,Y -623.923,Z 872.667,A 0.000,B 0.000,C 90.000,E1 336.049} C_DIS
LIN {X -0.180,Y -628.493,Z 872.661,A 0.000,B 0.000,C 90.000,E1 335.049} C_DIS
LIN {X -0.115,Y -631.642,Z 872.657,A 0.000,B 0.000,C 90.000,E1 334.280} C_DIS
LIN {X 0.026,Y -635.659,Z 872.651,A 0.000,B 0.000,C 90.000,E1 333.256} C_DIS
LIN {X 0.221,Y -639.417,Z 872.646,A 0.000,B 0.000,C 90.000,E1 332.231} C_DIS
LIN {X -0.039,Y -643.756,Z 872.639,A 0.000,B 0.000,C 90.000,E1 331.001} C_DIS
LIN {X 0.007,Y -646.975,Z 872.633,A 0.000,B 0.000,C 90.000,E1 329.999} C_DIS
LIN {X 0.185,Y -650.770,Z 872.626,A 0.000,B 0.000,C 90.000,E1 328.742} C_DIS
LIN {X -0.228,Y -653.571,Z 872.621,A 0.000,B 0.000,C 90.000,E1 327.788} C_DIS
LIN {X -0.147,Y -656.805,Z 872.614,A 0.000,B 0.000,C 90.000,E1 326.548} C_DIS
LIN {X -0.012,Y -659.611,Z 872.607,A 0.000,B 0.000,C 90.000,E1 325.308} C_DIS
LIN {X 0.158,Y -661.942,Z 872.601,A 0.000,B 0.000,C 90.000,E1 324.069} C_DIS
LIN {X -0.277,Y -663.582,Z 872.595,A 0.000,B 0.000,C 90.000,E1 323.130} C_DIS
LIN {X 0.306,Y -665.668,Z 872.587,A 0.000,B 0.000,C 90.000,E1 321.618} C_DIS
LIN {X 0.393,Y -667.715,Z 872.578,A 0.000,B 0.000,C 90.000,E1 319.908} C_DIS
LIN {X 0.012,Y -669.083,Z 872.571,A 0.000,B 0.000,C 90.000,E1 318.728} C_DIS
LIN {X -0.403,Y -670.568,Z 872.563,A 0.000,B 0.000,C 90.000,E1 317.310} C_DIS
LIN {X 0.207,Y -672.866,Z 872.552,A 0.000,B 0.000,C 90.000,E1 315.324} C_DIS
LIN {X 0.272,Y -673.650,Z 872.548,A 0.000,B 0.000,C 90.000,E1 314.595} C_DIS
LIN {X 0.034,Y -675.707,Z 872.536,A 0.000,B 0.000,C 90.000,E1 312.447} C_DIS
LIN {X 0.248,Y -677.106,Z 872.528,A 0.000,B 0.000,C 90.000,E1 310.987} C_DIS
LIN {X -0.336,Y -678.713,Z 872.517,A 0.000,B 0.000,C 90.000,E1 309.116} C_DIS
LIN {X -0.006,Y -679.679,Z 872.511,A 0.000,B 0.000,C 90.000,E1 307.890} C_DIS
LIN {X -0.199,Y -680.627,Z 872.504,A 0.000,B 0.000,C 90.000,E1 306.710} C_DIS
LIN {X 0.320,Y -681.640,Z 872.496,A 0.000,B 0.000,C 90.000,E1 305.231} C_DIS
LIN {X -0.092,Y -682.526,Z 872.488,A 0.000,B 0.000,C 90.000,E1 303.833} C_DIS
LIN {X -0.293,Y -683.506,Z 872.480,A 0.000,B 0.000,C 90.000,E1 302.418} C_DIS
LIN {X 0.093,Y -684.782,Z 872.471,A 0.000,B 0.000,C 90.000,E1 300.718} C_DIS
LIN {X -0.033,Y -685.761,Z 872.464,A 0.000,B 0.000,C 90.000,E1 299.539} C_DIS
LIN {X 0.085,Y -687.111,Z 872.456,A 0.000,B 0.000,C 90.000,E1 298.103} C_DIS
LIN {X -0.087,Y -688.617,Z 872.448,A 0.000,B 0.000,C 90.000,E1 296.693} C_DIS
LIN {X -0.229,Y -690.163,Z 872.440,A 0.000,B 0.000,C 90.000,E1 295.283} C_DIS
LIN {X -0.201,Y -691.033,Z 872.435,A 0.000,B 0.000,C 90.000,E1 294.335} C_DIS
LIN {X 0.272,Y -691.347,Z 872.432,A 0.000,B 0.000,C 90.000,E1 293.823} C_DIS
LIN {X -0.167,Y -691.486,Z 872.430,A 0.000,B 0.000,C 90.000,E1 293.387} C_DIS
LIN {X 0.032,Y -690.962,Z 872.427,A 0.000,B 0.000,C 90.000,E1 292.898} C_DIS
LIN {X 0.266,Y -690.565,Z 872.426,A 0.000,B 0.000,C 90.000,E1 292.642} C_DIS
LIN {X -0.175,Y -688.411,Z 872.423,A 0.000,B 0.000,C 90.000,E1 292.206} C_DIS
LIN {X -0.208,Y -687.050,Z 872.422,A 0.000,B 0.000,C 90.000,E1 291.972} C_DIS
LIN {X -0.099,Y -685.960,Z 872.421,A 0.000,B 0.000,C 90.000,E1 291.844} C_DIS
LIN {X 0.010,Y -684.317,Z 872.421,A 0.000,B 0.000,C 90.000,E1 291.716} C_DIS
LIN {X 0.185,Y -679.543,Z 872.419,A 0.000,B 0.000,C 90.000,E1 291.408} C_DIS
LIN {X -0.274,Y -677.813,Z 872.419,A 0.000,B 0.000,C 90.000,E1 291.354} C_DIS
LIN {X 0.251,Y -675.487,Z 872.418,A 0.000,B 0.000,C 90.000,E1 291.227} C_DIS
LIN {X 0.220,Y -669.043,Z 872.417,A 0.000,B 0.000,C 90.000,E1 291.046} C_DIS
LIN {X 0.192,Y -661.482,Z 872.416,A 0.000,B 0.000,C 90.000,E1 290.865} C_DIS
LIN {X -0.342,Y -656.463,Z 872.415,A 0.000,B 0.000,C 90.000,E1 290.737} C_DIS
LIN {X -0.150,Y -652.855,Z 872.414,A 0.000,B 0.000,C 90.000,E1 290.556} C_DIS
LIN {X -0.031,Y -650.564,Z 872.413,A 0.000,B 0.000,C 90.000,E1 290.355} C_DIS
LIN {X -0.072,Y -650.539,Z 872.413,A 0.000,B 0.000,C 90.000,E1 290.355} C_DIS
LIN {X 0.088,Y -650.363,Z 872.413,A 0.000,B 0.000,C 90.000,E1 290.248} C_DIS
LIN {X 0.142,Y -651.394,Z 872.410,A 0.000,B 0.000,C 90.000,E1 289.812} C_DIS
LIN {X -0.095,Y -654.354,Z 872.407,A 0.000,B 0.000,C 90.000,E1 289.214} C_DIS
LIN {X -0.162,Y -659.583,Z 872.401,A 0.000,B 0.000,C 90.000,E1 288.236} C_DIS
LIN {X -0.328,Y -662.646,Z 872.398,A 0.000,B 0.000,C 90.000,E1 287.638} C_DIS
LIN {X 0.258,Y -664.408,Z 872.396,A 0.000,B 0.000,C 90.000,E1 287.221} C_DIS
LIN {X 0.184,Y -667.435,Z 872.392,A 0.000,B 0.000,C 90.000,E1 286.496} C_DIS
LIN {X -0.050,Y -669.913,Z 872.388,A 0.000,B 0.000,C 90.000,E1 285.788} C_DIS
LIN {X -0.012,Y -671.350,Z 872.385,A 0.000,B 0.000,C 90.000,E1 285.300} C_DIS
LIN {X -0.146,Y -672.548,Z 872.382,A 0.000,B 0.000,C 90.000,E1 284.828} C_DIS
LIN {X 0.324,Y -673.909,Z 872.378,A 0.000,B 0.000,C 90.000,E1 284.064} C_DIS
LIN {X 0.211,Y -674.697,Z 872.376,A 0.000,B 0.000,C 90.000,E1 283.592} C_DIS
LIN {X -0.005,Y -675.733,Z 872.370,A 0.000,B 0.000,C 90.000,E1 282.647} C_DIS
LIN {X -0.303,Y -676.245,Z 872.366,A 0.000,B 0.000,C 90.000,E1 281.951} C_DIS
LIN {X 0.259,Y -676.310,Z 872.364,A 0.000,B 0.000,C 90.000,E1 281.422} C_DIS
LIN {X 0.101,Y -676.011,Z 872.360,A 0.000,B 0.000,C 90.000,E1 280.715} C_DIS
LIN {X -0.131,Y -675.564,Z 872.357,A 0.000,B 0.000,C 90.000,E1 280.254} C_DIS
LIN {X -0.247,Y -674.824,Z 872.354,A 0.000,B 0.000,C 90.000,E1 279.782} C_DIS
LIN {X 0.183,Y -673.801,Z 872.352,A 0.000,B 0.000,C 90.000,E1 279.265} C_DIS
LIN {X -0.054,Y -672.440,Z 872.349,A 0.000,B 0.000,C 90.000,E1 278.803} C_DIS
LIN {X -0.295,Y -670.782,Z 872.346,A 0.000,B 0.000,C 90.000,E1 278.341} C_DIS
LIN {X 0.292,Y -669.897,Z 872.345,A 0.000,B 0.000,C 90.000,E1 278.049} C_DIS
LIN {X 0.036,Y -667.795,Z 872.342,A 0.000,B 0.000,C 90.000,E1 277.587} C_DIS
LIN {X -0.241,Y -664.786,Z 872.339,A 0.000,B 0.000,C 90.000,E1 277.004} C_DIS
LIN {X 0.032,Y -661.262,Z 872.335,A 0.000,B 0.000,C 90.000,E1 276.372} C_DIS
LIN {X -0.282,Y -658.010,Z 872.333,A 0.000,B 0.000,C 90.000,E1 275.910} C_DIS
LIN {X 0.036,Y -654.323,Z 872.330,A 0.000,B 0.000,C 90.000,E1 275.391} C_DIS
LIN {X 0.215,Y -648.758,Z 872.327,A 0.000,B 0.000,C 90.000,E1 274.759} C_DIS
LIN {X -0.163,Y -643.902,Z 872.324,A 0.000,B 0.000,C 90.000,E1 274.302} C_DIS
LIN {X 0.305,Y -637.325,Z 872.321,A 0.000,B 0.000,C 90.000,E1 273.669} C_DIS
LIN {X -0.125,Y -630.486,Z 872.318,A 0.000,B 0.000,C 90.000,E1 273.154} C_DIS
LIN {X 0.261,Y -624.557,Z 872.315,A 0.000,B 0.000,C 90.000,E1 272.694} C_DIS
LIN {X -0.263,Y -618.365,Z 872.313,A 0.000,B 0.000,C 90.000,E1 272.350} C_DIS
LIN {X -0.219,Y -610.204,Z 872.310,A 0.000,B 0.000,C 90.000,E1 271.892} C_DIS
LIN {X -0.034,Y -603.276,Z 872.309,A 0.000,B 0.000,C 90.000,E1 271.547} C_DIS
LIN {X 0.052,Y -598.029,Z 872.307,A 0.000,B 0.000,C 90.000,E1 271.318} C_DIS
LIN {X -0.268,Y -590.905,Z 872.306,A 0.000,B 0.000,C 90.000,E1 271.088} C_DIS
LIN {X -0.144,Y -583.623,Z 872.305,A 0.000,B 0.000,C 90.000,E1 270.859} C_DIS
LIN {X 0.267,Y -577.898,Z 872.304,A 0.000,B 0.000,C 90.000,E1 270.688} C_DIS
LIN {X 0.252,Y -571.551,Z 872.303,A 0.000,B 0.000,C 90.000,E1 270.573} C_DIS
LIN {X 0.016,Y -564.105,Z 872.303,A 0.000,B 0.000,C 90.000,E1 270.516} C_DIS
LIN {X -0.140,Y -552.331,Z 872.302,A 0.000,B 0.000,C 90.000,E1 270.458} C_DIS
LIN {X 0.270,Y -550.004,Z 872.302,A 0.000,B 0.000,C 90.000,E1 270.344} C_DIS
LIN {X 0.240,Y -549.924,Z 872.302,A 0.000,B 0.000,C 90.000,E1 270.344} C_DIS
LIN {X 0.115,Y -548.482,Z 872.301,A 0.000,B 0.000,C 90.000,E1 270.172} C_DIS
LIN {X 0.122,Y -546.928,Z 872.300,A 0.000,B 0.000,C 90.000,E1 270.000} C_DIS
LIN {X 0.080,Y -546.894,Z 872.300,A 0.000,B 0.000,C 90.000,E1 270.000} C_DIS
LIN {X -0.081,Y -546.232,Z 872.299,A 0.000,B 0.000,C 90.000,E1 269.771} C_DIS
LIN {X 0.081,Y -544.757,Z 872.292,A 0.000,B 0.000,C 90.000,E1 268.625} C_DIS
LIN {X -0.137,Y -542.638,Z 872.278,A 0.000,B 0.000,C 90.000,E1 266.102} C_DIS
LIN {X 0.046,Y -541.721,Z 872.270,A 0.000,B 0.000,C 90.000,E1 264.666} C_DIS
LIN {X 0.196,Y -540.910,Z 872.264,A 0.000,B 0.000,C 90.000,E1 263.514} C_DIS
LIN {X -0.134,Y -540.013,Z 872.258,A 0.000,B 0.000,C 90.000,E1 262.413} C_DIS
LIN {X 0.118,Y -538.478,Z 872.248,A 0.000,B 0.000,C 90.000,E1 260.679} C_DIS
LIN {X -0.121,Y -536.726,Z 872.239,A 0.000,B 0.000,C 90.000,E1 258.993} C_DIS
LIN {X -0.181,Y -534.842,Z 872.229,A 0.000,B 0.000,C 90.000,E1 257.285} C_DIS
LIN {X 0.027,Y -533.433,Z 872.223,A 0.000,B 0.000,C 90.000,E1 256.117} C_DIS
LIN {X 0.032,Y -531.285,Z 872.213,A 0.000,B 0.000,C 90.000,E1 254.393} C_DIS
LIN {X -0.011,Y -529.264,Z 872.204,A 0.000,B 0.000,C 90.000,E1 252.670} C_DIS
LIN {X 0.031,Y -527.921,Z 872.197,A 0.000,B 0.000,C 90.000,E1 251.511} C_DIS
LIN {X 0.234,Y -525.631,Z 872.188,A 0.000,B 0.000,C 90.000,E1 249.752} C_DIS
LIN {X -0.090,Y -523.640,Z 872.180,A 0.000,B 0.000,C 90.000,E1 248.337} C_DIS
LIN {X -0.297,Y -521.035,Z 872.170,A 0.000,B 0.000,C 90.000,E1 246.613} C_DIS
LIN {X 0.035,Y -519.268,Z 872.163,A 0.000,B 0.000,C 90.000,E1 245.409} C_DIS
LIN {X 0.014,Y -517.014,Z 872.155,A 0.000,B 0.000,C 90.000,E1 243.948} C_DIS
LIN {X -0.173,Y -515.048,Z 872.149,A 0.000,B 0.000,C 90.000,E1 242.794} C_DIS
LIN {X 0.055,Y -511.986,Z 872.139,A 0.000,B 0.000,C 90.000,E1 241.001} C_DIS
LIN {X -0.079,Y -509.402,Z 872.131,A 0.000,B 0.000,C 90.000,E1 239.537} C_DIS
LIN {X 0.008,Y -506.663,Z 872.122,A 0.000,B 0.000,C 90.000,E1 238.043} C_DIS
LIN {X 0.051,Y -503.822,Z 872.114,A 0.000,B 0.000,C 90.000,E1 236.548} C_DIS
LIN {X -0.266,Y -501.375,Z 872.108,A 0.000,B 0.000,C 90.000,E1 235.388} C_DIS
LIN {X -0.060,Y -497.808,Z 872.099,A 0.000,B 0.000,C 90.000,E1 233.863} C_DIS
LIN {X -0.035,Y -494.186,Z 872.091,A 0.000,B 0.000,C 90.000,E1 232.351} C_DIS
LIN {X 0.229,Y -490.654,Z 872.082,A 0.000,B 0.000,C 90.000,E1 230.803} C_DIS
LIN {X -0.120,Y -486.459,Z 872.072,A 0.000,B 0.000,C 90.000,E1 229.013} C_DIS
LIN {X 0.132,Y -483.685,Z 872.065,A 0.000,B 0.000,C 90.000,E1 227.757} C_DIS
LIN {X 0.145,Y -480.362,Z 872.057,A 0.000,B 0.000,C 90.000,E1 226.215} C_DIS
LIN {X 0.191,Y -476.373,Z 872.047,A 0.000,B 0.000,C 90.000,E1 224.352} C_DIS
LIN {X -0.095,Y -471.480,Z 872.034,A 0.000,B 0.000,C 90.000,E1 222.204} C_DIS
LIN {X -0.129,Y -466.688,Z 872.022,A 0.000,B 0.000,C 90.000,E1 220.011} C_DIS
LIN {X -0.224,Y -461.973,Z 872.010,A 0.000,B 0.000,C 90.000,E1 217.810} C_DIS
LIN {X 0.166,Y -458.672,Z 872.001,A 0.000,B 0.000,C 90.000,E1 216.171} C_DIS
LIN {X -0.048,Y -454.615,Z 871.990,A 0.000,B 0.000,C 90.000,E1 214.278} C_DIS
LIN {X 0.183,Y -449.122,Z 871.976,A 0.000,B 0.000,C 90.000,E1 211.671} C_DIS
LIN {X 0.019,Y -444.915,Z 871.965,A 0.000,B 0.000,C 90.000,E1 209.745} C_DIS
LIN {X 0.092,Y -441.476,Z 871.956,A 0.000,B 0.000,C 90.000,E1 208.103} C_DIS
LIN {X -0.084,Y -437.201,Z 871.945,A 0.000,B 0.000,C 90.000,E1 206.155} C_DIS
LIN {X 0.001,Y -434.383,Z 871.938,A 0.000,B 0.000,C 90.000,E1 204.823} C_DIS
LIN {X 0.079,Y -430.946,Z 871.929,A 0.000,B 0.000,C 90.000,E1 203.153} C_DIS
LIN {X 0.101,Y -427.565,Z 871.919,A 0.000,B 0.000,C 90.000,E1 201.482} C_DIS
LIN {X -0.163,Y -423.453,Z 871.908,A 0.000,B 0.000,C 90.000,E1 199.504} C_DIS
LIN {X -0.188,Y -420.161,Z 871.899,A 0.000,B 0.000,C 90.000,E1 197.819} C_DIS
LIN {X -0.037,Y -417.498,Z 871.891,A 0.000,B 0.000,C 90.000,E1 196.441} C_DIS
LIN {X -0.158,Y -413.295,Z 871.880,A 0.000,B 0.000,C 90.000,E1 194.411} C_DIS
LIN {X -0.186,Y -409.293,Z 871.869,A 0.000,B 0.000,C 90.000,E1 192.355} C_DIS
LIN {X -0.006,Y -405.957,Z 871.859,A 0.000,B 0.000,C 90.000,E1 190.602} C_DIS
LIN {X 0.034,Y -402.484,Z 871.849,A 0.000,B 0.000,C 90.000,E1 188.859} C_DIS
LIN {X -0.054,Y -398.961,Z 871.840,A 0.000,B 0.000,C 90.000,E1 187.125} C_DIS
LIN {X -0.052,Y -393.195,Z 871.822,A 0.000,B 0.000,C 90.000,E1 183.955} C_DIS
LIN {X -0.187,Y -389.426,Z 871.808,A 0.000,B 0.000,C 90.000,E1 181.489} C_DIS
LIN {X 0.045,Y -386.404,Z 871.796,A 0.000,B 0.000,C 90.000,E1 179.312} C_DIS
LIN {X -0.069,Y -383.777,Z 871.786,A 0.000,B 0.000,C 90.000,E1 177.535} C_DIS
LIN {X 0.165,Y -381.143,Z 871.776,A 0.000,B 0.000,C 90.000,E1 175.698} C_DIS
LIN {X -0.143,Y -378.061,Z 871.764,A 0.000,B 0.000,C 90.000,E1 173.571} C_DIS
LIN {X -0.180,Y -375.092,Z 871.750,A 0.000,B 0.000,C 90.000,E1 171.027} C_DIS
LIN {X 0.061,Y -373.647,Z 871.740,A 0.000,B 0.000,C 90.000,E1 169.162} C_DIS
LIN {X 0.149,Y -373.403,Z 871.734,A 0.000,B 0.000,C 90.000,E1 168.049} C_DIS
LIN {X 0.112,Y -373.645,Z 871.726,A 0.000,B 0.000,C 90.000,E1 166.589} C_DIS
LIN {X 0.064,Y -374.129,Z 871.722,A 0.000,B 0.000,C 90.000,E1 165.992} C_DIS
LIN {X -0.043,Y -374.247,Z 871.721,A 0.000,B 0.000,C 90.000,E1 165.825} C_DIS
LIN {X -0.102,Y -374.953,Z 871.719,A 0.000,B 0.000,C 90.000,E1 165.408} C_DIS
LIN {X -0.130,Y -375.345,Z 871.717,A 0.000,B 0.000,C 90.000,E1 165.046} C_DIS
LIN {X 0.209,Y -376.321,Z 871.715,A 0.000,B 0.000,C 90.000,E1 164.629} C_DIS
LIN {X 0.087,Y -377.030,Z 871.713,A 0.000,B 0.000,C 90.000,E1 164.283} C_DIS
LIN {X 0.063,Y -379.151,Z 871.710,A 0.000,B 0.000,C 90.000,E1 163.740} C_DIS
LIN {X -0.180,Y -379.910,Z 871.708,A 0.000,B 0.000,C 90.000,E1 163.504} C_DIS
LIN {X 0.053,Y -382.659,Z 871.706,A 0.000,B 0.000,C 90.000,E1 163.015} C_DIS
LIN {X -0.086,Y -386.110,Z 871.703,A 0.000,B 0.000,C 90.000,E1 162.598} C_DIS
LIN {X -0.022,Y -387.798,Z 871.702,A 0.000,B 0.000,C 90.000,E1 162.417} C_DIS
LIN {X 0.147,Y -393.029,Z 871.700,A 0.000,B 0.000,C 90.000,E1 162.000} C_DIS
LIN {X 0.009,Y -399.086,Z 871.698,A 0.000,B 0.000,C 90.000,E1 161.692} C_DIS
LIN {X 0.099,Y -412.874,Z 871.695,A 0.000,B 0.000,C 90.000,E1 161.040} C_DIS
LIN {X 0.026,Y -414.654,Z 871.694,A 0.000,B 0.000,C 90.000,E1 160.967} C_DIS
LIN {X -0.021,Y -424.202,Z 871.691,A 0.000,B 0.000,C 90.000,E1 160.423} C_DIS
LIN {X 0.000,Y -430.812,Z 871.689,A 0.000,B 0.000,C 90.000,E1 160.007} C_DIS
LIN {X 0.073,Y -437.223,Z 871.687,A 0.000,B 0.000,C 90.000,E1 159.571} C_DIS
LIN {X -0.098,Y -441.690,Z 871.685,A 0.000,B 0.000,C 90.000,E1 159.263} C_DIS
LIN {X 0.008,Y -449.452,Z 871.681,A 0.000,B 0.000,C 90.000,E1 158.646} C_DIS
LIN {X -0.118,Y -453.914,Z 871.679,A 0.000,B 0.000,C 90.000,E1 158.284} C_DIS
LIN {X 0.225,Y -458.377,Z 871.677,A 0.000,B 0.000,C 90.000,E1 157.847} C_DIS
LIN {X 0.133,Y -469.645,Z 871.671,A 0.000,B 0.000,C 90.000,E1 156.741} C_DIS
LIN {X 0.016,Y -475.081,Z 871.668,A 0.000,B 0.000,C 90.000,E1 156.177} C_DIS
LIN {X 0.166,Y -481.653,Z 871.664,A 0.000,B 0.000,C 90.000,E1 155.409} C_DIS
LIN {X 0.038,Y -488.066,Z 871.659,A 0.000,B 0.000,C 90.000,E1 154.665} C_DIS
LIN {X -0.122,Y -495.370,Z 871.654,A 0.000,B 0.000,C 90.000,E1 153.768} C_DIS
LIN {X -0.060,Y -498.839,Z 871.652,A 0.000,B 0.000,C 90.000,E1 153.307} C_DIS
LIN {X 0.156,Y -506.584,Z 871.646,A 0.000,B 0.000,C 90.000,E1 152.231} C_DIS
LIN {X 0.086,Y -514.930,Z 871.639,A 0.000,B 0.000,C 90.000,E1 151.051} C_DIS
LIN {X -0.241,Y -521.184,Z 871.634,A 0.000,B 0.000,C 90.000,E1 150.205} C_DIS
LIN {X -0.083,Y -525.647,Z 871.630,A 0.000,B 0.000,C 90.000,E1 149.459} C_DIS
LIN {X 0.007,Y -529.393,Z 871.627,A 0.000,B 0.000,C 90.000,E1 148.869} C_DIS
LIN {X 0.101,Y -534.549,Z 871.622,A 0.000,B 0.000,C 90.000,E1 147.995} C_DIS
LIN {X 0.106,Y -540.316,Z 871.617,A 0.000,B 0.000,C 90.000,E1 146.993} C_DIS
LIN {X -0.140,Y -545.117,Z 871.612,A 0.000,B 0.000,C 90.000,E1 146.167} C_DIS
LIN {X -0.027,Y -549.598,Z 871.607,A 0.000,B 0.000,C 90.000,E1 145.308} C_DIS
LIN {X -0.175,Y -554.039,Z 871.603,A 0.000,B 0.000,C 90.000,E1 144.482} C_DIS
LIN {X 0.044,Y -558.263,Z 871.598,A 0.000,B 0.000,C 90.000,E1 143.623} C_DIS
LIN {X -0.373,Y -563.962,Z 871.592,A 0.000,B 0.000,C 90.000,E1 142.557} C_DIS
LIN {X -0.003,Y -571.624,Z 871.583,A 0.000,B 0.000,C 90.000,E1 141.009} C_DIS
LIN {X 0.112,Y -577.087,Z 871.577,A 0.000,B 0.000,C 90.000,E1 139.908} C_DIS
LIN {X 0.130,Y -582.757,Z 871.571,A 0.000,B 0.000,C 90.000,E1 138.690} C_DIS
LIN {X -0.307,Y -593.655,Z 871.558,A 0.000,B 0.000,C 90.000,E1 136.458} C_DIS
LIN {X -0.236,Y -595.626,Z 871.556,A 0.000,B 0.000,C 90.000,E1 136.053} C_DIS
LIN {X -0.064,Y -601.820,Z 871.548,A 0.000,B 0.000,C 90.000,E1 134.717} C_DIS
LIN {X 0.032,Y -609.108,Z 871.540,A 0.000,B 0.000,C 90.000,E1 133.137} C_DIS
LIN {X 0.026,Y -614.782,Z 871.532,A 0.000,B 0.000,C 90.000,E1 131.838} C_DIS
LIN {X -0.186,Y -619.224,Z 871.527,A 0.000,B 0.000,C 90.000,E1 130.825} C_DIS
LIN {X 0.054,Y -624.391,Z 871.520,A 0.000,B 0.000,C 90.000,E1 129.519} C_DIS
LIN {X -0.234,Y -630.261,Z 871.511,A 0.000,B 0.000,C 90.000,E1 128.016} C_DIS
LIN {X -0.177,Y -635.096,Z 871.504,A 0.000,B 0.000,C 90.000,E1 126.744} C_DIS
LIN {X -0.048,Y -638.814,Z 871.498,A 0.000,B 0.000,C 90.000,E1 125.724} C_DIS
LIN {X -0.125,Y -641.424,Z 871.494,A 0.000,B 0.000,C 90.000,E1 124.978} C_DIS
LIN {X -0.291,Y -644.615,Z 871.489,A 0.000,B 0.000,C 90.000,E1 123.992} C_DIS
LIN {X 0.117,Y -647.562,Z 871.483,A 0.000,B 0.000,C 90.000,E1 122.959} C_DIS
LIN {X 0.137,Y -649.492,Z 871.479,A 0.000,B 0.000,C 90.000,E1 122.212} C_DIS
LIN {X -0.292,Y -651.788,Z 871.474,A 0.000,B 0.000,C 90.000,E1 121.258} C_DIS
LIN {X 0.324,Y -653.349,Z 871.469,A 0.000,B 0.000,C 90.000,E1 120.463} C_DIS
LIN {X -0.286,Y -655.558,Z 871.463,A 0.000,B 0.000,C 90.000,E1 119.283} C_DIS
LIN {X 0.144,Y -655.998,Z 871.461,A 0.000,B 0.000,C 90.000,E1 118.999} C_DIS
LIN {X -0.195,Y -658.603,Z 871.452,A 0.000,B 0.000,C 90.000,E1 117.308} C_DIS
LIN {X 0.015,Y -660.061,Z 871.446,A 0.000,B 0.000,C 90.000,E1 116.309} C_DIS
LIN {X -0.053,Y -661.078,Z 871.441,A 0.000,B 0.000,C 90.000,E1 115.335} C_DIS
LIN {X 0.337,Y -661.788,Z 871.434,A 0.000,B 0.000,C 90.000,E1 114.079} C_DIS
LIN {X -0.136,Y -661.769,Z 871.433,A 0.000,B 0.000,C 90.000,E1 113.875} C_DIS
LIN {X -0.136,Y -661.160,Z 871.430,A 0.000,B 0.000,C 90.000,E1 113.387} C_DIS
LIN {X -0.006,Y -660.493,Z 871.429,A 0.000,B 0.000,C 90.000,E1 113.131} C_DIS
LIN {X -0.009,Y -658.547,Z 871.426,A 0.000,B 0.000,C 90.000,E1 112.642} C_DIS
LIN {X 0.111,Y -656.689,Z 871.424,A 0.000,B 0.000,C 90.000,E1 112.386} C_DIS
LIN {X 0.030,Y -653.518,Z 871.422,A 0.000,B 0.000,C 90.000,E1 112.025} C_DIS
LIN {X 0.210,Y -647.206,Z 871.420,A 0.000,B 0.000,C 90.000,E1 111.589} C_DIS
LIN {X -0.303,Y -645.510,Z 871.420,A 0.000,B 0.000,C 90.000,E1 111.535} C_DIS
LIN {X -0.053,Y -640.626,Z 871.419,A 0.000,B 0.000,C 90.000,E1 111.334} C_DIS
LIN {X 0.333,Y -636.522,Z 871.417,A 0.000,B 0.000,C 90.000,E1 111.099} C_DIS
LIN {X 0.041,Y -627.570,Z 871.416,A 0.000,B 0.000,C 90.000,E1 110.791} C_DIS
LIN {X -0.054,Y -614.391,Z 871.413,A 0.000,B 0.000,C 90.000,E1 110.301} C_DIS
LIN {X -0.254,Y -606.833,Z 871.411,A 0.000,B 0.000,C 90.000,E1 109.993} C_DIS
LIN {X 0.173,Y -593.792,Z 871.408,A 0.000,B 0.000,C 90.000,E1 109.341} C_DIS
LIN {X 0.187,Y -586.998,Z 871.406,A 0.000,B 0.000,C 90.000,E1 109.033} C_DIS
LIN {X 0.076,Y -579.742,Z 871.404,A 0.000,B 0.000,C 90.000,E1 108.779} C_DIS
LIN {X -0.134,Y -567.137,Z 871.402,A 0.000,B 0.000,C 90.000,E1 108.417} C_DIS
LIN {X 0.075,Y -564.950,Z 871.402,A 0.000,B 0.000,C 90.000,E1 108.308} C_DIS
LIN {X -0.026,Y -562.170,Z 871.401,A 0.000,B 0.000,C 90.000,E1 108.181} C_DIS
LIN {X 0.014,Y -560.417,Z 871.400,A 0.000,B 0.000,C 90.000,E1 108.000} C_DIS
LIN {X 0.011,Y -560.089,Z 871.400,A 0.000,B 0.000,C 90.000,E1 107.946} C_DIS
LIN {X -0.220,Y -558.969,Z 871.398,A 0.000,B 0.000,C 90.000,E1 107.692} C_DIS
LIN {X -0.089,Y -558.560,Z 871.397,A 0.000,B 0.000,C 90.000,E1 107.402} C_DIS
LIN {X 0.205,Y -558.348,Z 871.395,A 0.000,B 0.000,C 90.000,E1 107.094} C_DIS
LIN {X 0.142,Y -559.467,Z 871.372,A 0.000,B 0.000,C 90.000,E1 102.939} C_DIS
LIN {X 0.074,Y -560.652,Z 871.361,A 0.000,B 0.000,C 90.000,E1 101.007} C_DIS
LIN {X -0.226,Y -561.840,Z 871.352,A 0.000,B 0.000,C 90.000,E1 99.378} C_DIS
LIN {X -0.033,Y -562.968,Z 871.343,A 0.000,B 0.000,C 90.000,E1 97.701} C_DIS
LIN {X 0.034,Y -563.834,Z 871.335,A 0.000,B 0.000,C 90.000,E1 96.315} C_DIS
LIN {X 0.056,Y -564.466,Z 871.328,A 0.000,B 0.000,C 90.000,E1 94.935} C_DIS
LIN {X 0.091,Y -565.041,Z 871.320,A 0.000,B 0.000,C 90.000,E1 93.555} C_DIS
LIN {X 0.101,Y -565.499,Z 871.312,A 0.000,B 0.000,C 90.000,E1 92.178} C_DIS
LIN {X 0.116,Y -565.958,Z 871.305,A 0.000,B 0.000,C 90.000,E1 90.802} C_DIS
LIN {X 0.243,Y -566.327,Z 871.295,A 0.000,B 0.000,C 90.000,E1 89.141} C_DIS
LIN {X -0.178,Y -566.614,Z 871.286,A 0.000,B 0.000,C 90.000,E1 87.535} C_DIS
LIN {X 0.005,Y -566.921,Z 871.277,A 0.000,B 0.000,C 90.000,E1 85.869} C_DIS
LIN {X 0.086,Y -567.147,Z 871.269,A 0.000,B 0.000,C 90.000,E1 84.489} C_DIS
LIN {X -0.232,Y -567.444,Z 871.260,A 0.000,B 0.000,C 90.000,E1 82.875} C_DIS
LIN {X 0.175,Y -567.993,Z 871.250,A 0.000,B 0.000,C 90.000,E1 80.914} C_DIS
LIN {X 0.203,Y -568.671,Z 871.239,A 0.000,B 0.000,C 90.000,E1 78.993} C_DIS
LIN {X -0.194,Y -569.563,Z 871.228,A 0.000,B 0.000,C 90.000,E1 77.117} C_DIS
LIN {X 0.113,Y -570.214,Z 871.218,A 0.000,B 0.000,C 90.000,E1 75.172} C_DIS
LIN {X 0.220,Y -570.658,Z 871.210,A 0.000,B 0.000,C 90.000,E1 73.795} C_DIS
LIN {X -0.002,Y -570.908,Z 871.204,A 0.000,B 0.000,C 90.000,E1 72.725} C_DIS
LIN {X 0.114,Y -571.153,Z 871.196,A 0.000,B 0.000,C 90.000,E1 71.348} C_DIS
LIN {X 0.197,Y -571.325,Z 871.184,A 0.000,B 0.000,C 90.000,E1 69.156} C_DIS
LIN {X -0.179,Y -571.371,Z 871.174,A 0.000,B 0.000,C 90.000,E1 67.283} C_DIS
LIN {X -0.205,Y -571.345,Z 871.166,A 0.000,B 0.000,C 90.000,E1 65.921} C_DIS
LIN {X -0.005,Y -571.204,Z 871.159,A 0.000,B 0.000,C 90.000,E1 64.537} C_DIS
LIN {X -0.073,Y -570.982,Z 871.151,A 0.000,B 0.000,C 90.000,E1 63.179} C_DIS
LIN {X -0.136,Y -570.627,Z 871.143,A 0.000,B 0.000,C 90.000,E1 61.820} C_DIS
LIN {X -0.211,Y -570.143,Z 871.136,A 0.000,B 0.000,C 90.000,E1 60.461} C_DIS
LIN {X 0.043,Y -569.785,Z 871.131,A 0.000,B 0.000,C 90.000,E1 59.616} C_DIS
LIN {X -0.157,Y -568.627,Z 871.122,A 0.000,B 0.000,C 90.000,E1 57.995} C_DIS
LIN {X -0.228,Y -568.263,Z 871.119,A 0.000,B 0.000,C 90.000,E1 57.454} C_DIS
LIN {X -0.185,Y -567.501,Z 871.115,A 0.000,B 0.000,C 90.000,E1 56.628} C_DIS
LIN {X -0.032,Y -566.252,Z 871.108,A 0.000,B 0.000,C 90.000,E1 55.515} C_DIS
LIN {X 0.103,Y -564.872,Z 871.102,A 0.000,B 0.000,C 90.000,E1 54.402} C_DIS
LIN {X -0.242,Y -563.267,Z 871.096,A 0.000,B 0.000,C 90.000,E1 53.336} C_DIS
LIN {X 0.074,Y -561.922,Z 871.092,A 0.000,B 0.000,C 90.000,E1 52.477} C_DIS
LIN {X -0.067,Y -560.423,Z 871.087,A 0.000,B 0.000,C 90.000,E1 51.662} C_DIS
LIN {X 0.213,Y -558.729,Z 871.082,A 0.000,B 0.000,C 90.000,E1 50.803} C_DIS
LIN {X 0.037,Y -556.735,Z 871.078,A 0.000,B 0.000,C 90.000,E1 49.989} C_DIS
LIN {X -0.161,Y -554.434,Z 871.073,A 0.000,B 0.000,C 90.000,E1 49.175} C_DIS
LIN {X -0.082,Y -552.808,Z 871.070,A 0.000,B 0.000,C 90.000,E1 48.609} C_DIS
LIN {X 0.046,Y -549.921,Z 871.065,A 0.000,B 0.000,C 90.000,E1 47.757} C_DIS
LIN {X 0.172,Y -545.641,Z 871.059,A 0.000,B 0.000,C 90.000,E1 46.620} C_DIS
LIN {X -0.176,Y -542.077,Z 871.054,A 0.000,B 0.000,C 90.000,E1 45.810} C_DIS
LIN {X 0.013,Y -538.629,Z 871.051,A 0.000,B 0.000,C 90.000,E1 45.081} C_DIS
LIN {X 0.170,Y -534.873,Z 871.047,A 0.000,B 0.000,C 90.000,E1 44.352} C_DIS
LIN {X -0.058,Y -532.493,Z 871.044,A 0.000,B 0.000,C 90.000,E1 43.947} C_DIS
LIN {X 0.037,Y -528.050,Z 871.040,A 0.000,B 0.000,C 90.000,E1 43.218} C_DIS
LIN {X 0.317,Y -524.316,Z 871.037,A 0.000,B 0.000,C 90.000,E1 42.609} C_DIS
LIN {X -0.021,Y -519.280,Z 871.033,A 0.000,B 0.000,C 90.000,E1 41.919} C_DIS
LIN {X 0.059,Y -516.091,Z 871.030,A 0.000,B 0.000,C 90.000,E1 41.472} C_DIS
LIN {X -0.135,Y -511.544,Z 871.027,A 0.000,B 0.000,C 90.000,E1 40.906} C_DIS
LIN {X -0.080,Y -504.167,Z 871.022,A 0.000,B 0.000,C 90.000,E1 40.011} C_DIS
LIN {X 0.075,Y -498.812,Z 871.019,A 0.000,B 0.000,C 90.000,E1 39.402} C_DIS
LIN {X -0.038,Y -491.932,Z 871.015,A 0.000,B 0.000,C 90.000,E1 38.705} C_DIS
LIN {X -0.297,Y -486.153,Z 871.012,A 0.000,B 0.000,C 90.000,E1 38.177} C_DIS
LIN {X -0.299,Y -478.998,Z 871.008,A 0.000,B 0.000,C 90.000,E1 37.523} C_DIS
LIN {X 0.053,Y -470.012,Z 871.004,A 0.000,B 0.000,C 90.000,E1 36.710} C_DIS
LIN {X -0.067,Y -460.681,Z 871.000,A 0.000,B 0.000,C 90.000,E1 35.964} C_DIS
LIN {X -0.087,Y -449.810,Z 870.995,A 0.000,B 0.000,C 90.000,E1 35.105} C_DIS
LIN {X 0.000,Y -431.243,Z 870.987,A 0.000,B 0.000,C 90.000,E1 33.627} C_DIS
LIN {X -0.102,Y -409.999,Z 870.977,A 0.000,B 0.000,C 90.000,E1 31.799} C_DIS
LIN {X 0.020,Y -402.803,Z 870.973,A 0.000,B 0.000,C 90.000,E1 31.082} C_DIS
LIN {X -0.074,Y -397.217,Z 870.969,A 0.000,B 0.000,C 90.000,E1 30.463} C_DIS
LIN {X -0.102,Y -394.331,Z 870.967,A 0.000,B 0.000,C 90.000,E1 30.079} C_DIS
LIN {X -0.084,Y -393.322,Z 870.966,A 0.000,B 0.000,C 90.000,E1 29.922} C_DIS
LIN {X 0.085,Y -391.552,Z 870.964,A 0.000,B 0.000,C 90.000,E1 29.539} C_DIS
LIN {X -0.070,Y -390.165,Z 870.961,A 0.000,B 0.000,C 90.000,E1 29.027} C_DIS
LIN {X -0.029,Y -389.456,Z 870.957,A 0.000,B 0.000,C 90.000,E1 28.309} C_DIS
LIN {X 0.189,Y -389.483,Z 870.952,A 0.000,B 0.000,C 90.000,E1 27.385} C_DIS
LIN {X -0.133,Y -392.065,Z 870.931,A 0.000,B 0.000,C 90.000,E1 23.515} C_DIS
LIN {X -0.035,Y -394.744,Z 870.915,A 0.000,B 0.000,C 90.000,E1 20.663} C_DIS
LIN {X -0.098,Y -396.577,Z 870.905,A 0.000,B 0.000,C 90.000,E1 18.906} C_DIS
LIN {X -0.091,Y -399.450,Z 870.891,A 0.000,B 0.000,C 90.000,E1 16.441} C_DIS
LIN {X 0.181,Y -402.094,Z 870.880,A 0.000,B 0.000,C 90.000,E1 14.300} C_DIS
LIN {X 0.019,Y -405.521,Z 870.866,A 0.000,B 0.000,C 90.000,E1 11.883} C_DIS
LIN {X 0.133,Y -409.776,Z 870.851,A 0.000,B 0.000,C 90.000,E1 9.095} C_DIS
LIN {X -0.077,Y -414.466,Z 870.835,A 0.000,B 0.000,C 90.000,E1 6.372} C_DIS
LIN {X 0.134,Y -419.577,Z 870.820,A 0.000,B 0.000,C 90.000,E1 3.612} C_DIS
LIN {X -0.005,Y -424.491,Z 870.807,A 0.000,B 0.000,C 90.000,E1 1.260} C_DIS
LIN {X -0.136,Y -429.486,Z 870.795,A 0.000,B 0.000,C 90.000,E1 359.141} C_DIS
LIN {X 0.009,Y -435.225,Z 870.782,A 0.000,B 0.000,C 90.000,E1 356.788} C_DIS
LIN {X 0.110,Y -439.458,Z 870.773,A 0.000,B 0.000,C 90.000,E1 355.122} C_DIS
LIN {X -0.031,Y -442.285,Z 870.768,A 0.000,B 0.000,C 90.000,E1 354.318} C_DIS
LIN {X -0.200,Y -444.325,Z 870.766,A 0.000,B 0.000,C 90.000,E1 353.913} C_DIS
LIN {X -0.144,Y -445.402,Z 870.765,A 0.000,B 0.000,C 90.000,E1 353.742} C_DIS
LIN {X -0.124,Y -448.772,Z 870.763,A 0.000,B 0.000,C 90.000,E1 353.394} C_DIS
LIN {X -0.050,Y -450.036,Z 870.763,A 0.000,B 0.000,C 90.000,E1 353.280} C_DIS
LIN {X 0.079,Y -455.482,Z 870.761,A 0.000,B 0.000,C 90.000,E1 352.932} C_DIS
LIN {X 0.195,Y -463.815,Z 870.759,A 0.000,B 0.000,C 90.000,E1 352.534} C_DIS
LIN {X 0.124,Y -470.382,Z 870.757,A 0.000,B 0.000,C 90.000,E1 352.243} C_DIS
LIN {X -0.251,Y -480.400,Z 870.754,A 0.000,B 0.000,C 90.000,E1 351.781} C_DIS
LIN {X 0.102,Y -490.123,Z 870.751,A 0.000,B 0.000,C 90.000,E1 351.197} C_DIS
LIN {X 0.067,Y -499.773,Z 870.748,A 0.000,B 0.000,C 90.000,E1 350.622} C_DIS
LIN {X -0.078,Y -510.848,Z 870.744,A 0.000,B 0.000,C 90.000,E1 349.926} C_DIS
LIN {X -0.061,Y -518.616,Z 870.741,A 0.000,B 0.000,C 90.000,E1 349.398} C_DIS
LIN {X -0.216,Y -526.276,Z 870.738,A 0.000,B 0.000,C 90.000,E1 348.870} C_DIS
LIN {X 0.036,Y -533.672,Z 870.735,A 0.000,B 0.000,C 90.000,E1 348.285} C_DIS
LIN {X -0.162,Y -542.352,Z 870.731,A 0.000,B 0.000,C 90.000,E1 347.589} C_DIS
LIN {X 0.164,Y -549.278,Z 870.728,A 0.000,B 0.000,C 90.000,E1 346.937} C_DIS
LIN {X 0.175,Y -555.878,Z 870.724,A 0.000,B 0.000,C 90.000,E1 346.297} C_DIS
LIN {X 0.298,Y -561.075,Z 870.721,A 0.000,B 0.000,C 90.000,E1 345.755} C_DIS
LIN {X 0.168,Y -566.033,Z 870.718,A 0.000,B 0.000,C 90.000,E1 345.227} C_DIS
LIN {X -0.160,Y -571.930,Z 870.714,A 0.000,B 0.000,C 90.000,E1 344.574} C_DIS
LIN {X -0.083,Y -579.629,Z 870.709,A 0.000,B 0.000,C 90.000,E1 343.614} C_DIS
LIN {X 0.257,Y -584.635,Z 870.705,A 0.000,B 0.000,C 90.000,E1 342.906} C_DIS
LIN {X 0.255,Y -589.291,Z 870.701,A 0.000,B 0.000,C 90.000,E1 342.236} C_DIS
LIN {X 0.051,Y -594.485,Z 870.697,A 0.000,B 0.000,C 90.000,E1 341.456} C_DIS
LIN {X -0.160,Y -600.003,Z 870.692,A 0.000,B 0.000,C 90.000,E1 340.550} C_DIS
LIN {X 0.180,Y -606.725,Z 870.685,A 0.000,B 0.000,C 90.000,E1 339.337} C_DIS
LIN {X 0.006,Y -614.305,Z 870.677,A 0.000,B 0.000,C 90.000,E1 337.922} C_DIS
LIN {X -0.334,Y -618.901,Z 870.672,A 0.000,B 0.000,C 90.000,E1 337.050} C_DIS
LIN {X 0.200,Y -622.655,Z 870.668,A 0.000,B 0.000,C 90.000,E1 336.230} C_DIS
LIN {X -0.049,Y -626.175,Z 870.664,A 0.000,B 0.000,C 90.000,E1 335.485} C_DIS
LIN {X 0.016,Y -630.598,Z 870.658,A 0.000,B 0.000,C 90.000,E1 334.460} C_DIS
LIN {X -0.096,Y -635.651,Z 870.651,A 0.000,B 0.000,C 90.000,E1 333.204} C_DIS
LIN {X 0.390,Y -639.433,Z 870.646,A 0.000,B 0.000,C 90.000,E1 332.153} C_DIS
LIN {X 0.138,Y -643.786,Z 870.639,A 0.000,B 0.000,C 90.000,E1 330.923} C_DIS
LIN {X 0.189,Y -647.035,Z 870.633,A 0.000,B 0.000,C 90.000,E1 329.921} C_DIS
LIN {X -0.047,Y -650.108,Z 870.628,A 0.000,B 0.000,C 90.000,E1 328.948} C_DIS
LIN {X 0.083,Y -653.017,Z 870.622,A 0.000,B 0.000,C 90.000,E1 327.946} C_DIS
LIN {X 0.146,Y -656.291,Z 870.615,A 0.000,B 0.000,C 90.000,E1 326.707} C_DIS
LIN {X -0.296,Y -658.083,Z 870.611,A 0.000,B 0.000,C 90.000,E1 326.008} C_DIS
LIN {X -0.178,Y -659.753,Z 870.607,A 0.000,B 0.000,C 90.000,E1 325.261} C_DIS
LIN {X -0.162,Y -662.113,Z 870.600,A 0.000,B 0.000,C 90.000,E1 324.036} C_DIS
LIN {X -0.057,Y -663.784,Z 870.595,A 0.000,B 0.000,C 90.000,E1 323.050} C_DIS
LIN {X 0.035,Y -665.563,Z 870.588,A 0.000,B 0.000,C 90.000,E1 321.823} C_DIS
LIN {X 0.135,Y -667.412,Z 870.580,A 0.000,B 0.000,C 90.000,E1 320.356} C_DIS
LIN {X 0.190,Y -668.835,Z 870.573,A 0.000,B 0.000,C 90.000,E1 319.138} C_DIS
LIN {X 0.272,Y -670.118,Z 870.566,A 0.000,B 0.000,C 90.000,E1 317.919} C_DIS
LIN {X -0.005,Y -673.203,Z 870.552,A 0.000,B 0.000,C 90.000,E1 315.283} C_DIS
LIN {X 0.057,Y -673.963,Z 870.548,A 0.000,B 0.000,C 90.000,E1 314.555} C_DIS
LIN {X -0.366,Y -674.300,Z 870.545,A 0.000,B 0.000,C 90.000,E1 314.109} C_DIS
LIN {X 0.281,Y -675.748,Z 870.537,A 0.000,B 0.000,C 90.000,E1 312.609} C_DIS
LIN {X -0.010,Y -677.164,Z 870.529,A 0.000,B 0.000,C 90.000,E1 311.191} C_DIS
LIN {X 0.302,Y -678.403,Z 870.521,A 0.000,B 0.000,C 90.000,E1 309.725} C_DIS
LIN {X 0.122,Y -679.617,Z 870.513,A 0.000,B 0.000,C 90.000,E1 308.302} C_DIS
LIN {X -0.315,Y -680.932,Z 870.504,A 0.000,B 0.000,C 90.000,E1 306.664} C_DIS
LIN {X 0.049,Y -681.810,Z 870.497,A 0.000,B 0.000,C 90.000,E1 305.438} C_DIS
LIN {X 0.205,Y -682.713,Z 870.489,A 0.000,B 0.000,C 90.000,E1 303.992} C_DIS
LIN {X 0.203,Y -684.025,Z 870.478,A 0.000,B 0.000,C 90.000,E1 302.084} C_DIS
LIN {X -0.338,Y -685.335,Z 870.469,A 0.000,B 0.000,C 90.000,E1 300.463} C_DIS
LIN {X 0.061,Y -687.452,Z 870.456,A 0.000,B 0.000,C 90.000,E1 298.052} C_DIS
LIN {X 0.212,Y -688.937,Z 870.448,A 0.000,B 0.000,C 90.000,E1 296.616} C_DIS
LIN {X 0.070,Y -690.466,Z 870.440,A 0.000,B 0.000,C 90.000,E1 295.207} C_DIS
LIN {X 0.050,Y -691.488,Z 870.434,A 0.000,B 0.000,C 90.000,E1 294.027} C_DIS
LIN {X -0.147,Y -691.676,Z 870.430,A 0.000,B 0.000,C 90.000,E1 293.334} C_DIS
LIN {X 0.325,Y -691.049,Z 870.427,A 0.000,B 0.000,C 90.000,E1 292.823} C_DIS
LIN {X -0.346,Y -690.563,Z 870.426,A 0.000,B 0.000,C 90.000,E1 292.642} C_DIS
LIN {X -0.262,Y -688.881,Z 870.424,A 0.000,B 0.000,C 90.000,E1 292.280} C_DIS
LIN {X -0.036,Y -687.505,Z 870.422,A 0.000,B 0.000,C 90.000,E1 292.025} C_DIS
LIN {X 0.074,Y -686.633,Z 870.422,A 0.000,B 0.000,C 90.000,E1 291.897} C_DIS
LIN {X 0.182,Y -685.339,Z 870.421,A 0.000,B 0.000,C 90.000,E1 291.770} C_DIS
LIN {X -0.200,Y -681.987,Z 870.420,A 0.000,B 0.000,C 90.000,E1 291.589} C_DIS
LIN {X -0.182,Y -678.581,Z 870.419,A 0.000,B 0.000,C 90.000,E1 291.408} C_DIS
LIN {X 0.316,Y -676.830,Z 870.418,A 0.000,B 0.000,C 90.000,E1 291.280} C_DIS
LIN {X 0.017,Y -669.931,Z 870.417,A 0.000,B 0.000,C 90.000,E1 291.099} C_DIS
LIN {X 0.185,Y -660.807,Z 870.416,A 0.000,B 0.000,C 90.000,E1 290.865} C_DIS
LIN {X -0.352,Y -655.709,Z 870.415,A 0.000,B 0.000,C 90.000,E1 290.737} C_DIS
LIN {X -0.156,Y -652.062,Z 870.414,A 0.000,B 0.000,C 90.000,E1 290.556} C_DIS
LIN {X -0.047,Y -649.938,Z 870.413,A 0.000,B 0.000,C 90.000,E1 290.375} C_DIS
LIN {X -0.085,Y -649.920,Z 870.413,A 0.000,B 0.000,C 90.000,E1 290.375} C_DIS
LIN {X 0.065,Y -649.507,Z 870.413,A 0.000,B 0.000,C 90.000,E1 290.248} C_DIS
LIN {X 0.021,Y -649.501,Z 870.413,A 0.000,B 0.000,C 90.000,E1 290.248} C_DIS
LIN {X 0.134,Y -650.269,Z 870.411,A 0.000,B 0.000,C 90.000,E1 289.885} C_DIS
LIN {X -0.340,Y -652.576,Z 870.408,A 0.000,B 0.000,C 90.000,E1 289.396} C_DIS
LIN {X 0.077,Y -659.155,Z 870.401,A 0.000,B 0.000,C 90.000,E1 288.127} C_DIS
LIN {X -0.039,Y -662.797,Z 870.397,A 0.000,B 0.000,C 90.000,E1 287.402} C_DIS
LIN {X -0.126,Y -665.957,Z 870.393,A 0.000,B 0.000,C 90.000,E1 286.677} C_DIS
LIN {X -0.192,Y -668.515,Z 870.389,A 0.000,B 0.000,C 90.000,E1 285.953} C_DIS
LIN {X 0.299,Y -670.039,Z 870.386,A 0.000,B 0.000,C 90.000,E1 285.426} C_DIS
LIN {X 0.095,Y -671.837,Z 870.382,A 0.000,B 0.000,C 90.000,E1 284.717} C_DIS
LIN {X -0.091,Y -673.151,Z 870.378,A 0.000,B 0.000,C 90.000,E1 284.008} C_DIS
LIN {X -0.208,Y -673.910,Z 870.375,A 0.000,B 0.000,C 90.000,E1 283.536} C_DIS
LIN {X 0.282,Y -674.691,Z 870.371,A 0.000,B 0.000,C 90.000,E1 282.771} C_DIS
LIN {X 0.119,Y -675.225,Z 870.367,A 0.000,B 0.000,C 90.000,E1 282.063} C_DIS
LIN {X -0.178,Y -675.354,Z 870.363,A 0.000,B 0.000,C 90.000,E1 281.366} C_DIS
LIN {X -0.287,Y -675.195,Z 870.360,A 0.000,B 0.000,C 90.000,E1 280.894} C_DIS
LIN {X 0.262,Y -674.774,Z 870.358,A 0.000,B 0.000,C 90.000,E1 280.366} C_DIS
LIN {X -0.038,Y -673.692,Z 870.354,A 0.000,B 0.000,C 90.000,E1 279.670} C_DIS
LIN {X -0.278,Y -672.641,Z 870.351,A 0.000,B 0.000,C 90.000,E1 279.208} C_DIS
LIN {X 0.144,Y -671.189,Z 870.348,A 0.000,B 0.000,C 90.000,E1 278.690} C_DIS
LIN {X -0.008,Y -669.457,Z 870.346,A 0.000,B 0.000,C 90.000,E1 278.219} C_DIS
LIN {X -0.269,Y -667.441,Z 870.343,A 0.000,B 0.000,C 90.000,E1 277.757} C_DIS
LIN {X 0.120,Y -665.137,Z 870.340,A 0.000,B 0.000,C 90.000,E1 277.239} C_DIS
LIN {X -0.073,Y -663.234,Z 870.338,A 0.000,B 0.000,C 90.000,E1 276.891} C_DIS
LIN {X 0.284,Y -660.416,Z 870.336,A 0.000,B 0.000,C 90.000,E1 276.372} C_DIS
LIN {X -0.036,Y -657.141,Z 870.333,A 0.000,B 0.000,C 90.000,E1 275.910} C_DIS
LIN {X 0.274,Y -653.391,Z 870.330,A 0.000,B 0.000,C 90.000,E1 275.391} C_DIS
LIN {X -0.254,Y -647.823,Z 870.327,A 0.000,B 0.000,C 90.000,E1 274.821} C_DIS
LIN {X 0.076,Y -642.922,Z 870.324,A 0.000,B 0.000,C 90.000,E1 274.302} C_DIS
LIN {X -0.095,Y -637.613,Z 870.321,A 0.000,B 0.000,C 90.000,E1 273.841} C_DIS
LIN {X -0.025,Y -632.152,Z 870.319,A 0.000,B 0.000,C 90.000,E1 273.383} C_DIS
LIN {X 0.045,Y -625.172,Z 870.316,A 0.000,B 0.000,C 90.000,E1 272.865} C_DIS
LIN {X -0.307,Y -617.497,Z 870.313,A 0.000,B 0.000,C 90.000,E1 272.407} C_DIS
LIN {X 0.088,Y -610.905,Z 870.311,A 0.000,B 0.000,C 90.000,E1 272.007} C_DIS
LIN {X 0.172,Y -604.009,Z 870.309,A 0.000,B 0.000,C 90.000,E1 271.661} C_DIS
LIN {X 0.082,Y -596.864,Z 870.308,A 0.000,B 0.000,C 90.000,E1 271.375} C_DIS
LIN {X -0.207,Y -591.328,Z 870.307,A 0.000,B 0.000,C 90.000,E1 271.203} C_DIS
LIN {X -0.154,Y -583.862,Z 870.305,A 0.000,B 0.000,C 90.000,E1 270.974} C_DIS
LIN {X -0.143,Y -576.005,Z 870.304,A 0.000,B 0.000,C 90.000,E1 270.802} C_DIS
LIN {X 0.277,Y -571.917,Z 870.304,A 0.000,B 0.000,C 90.000,E1 270.688} C_DIS
LIN {X -0.003,Y -564.451,Z 870.304,A 0.000,B 0.000,C 90.000,E1 270.630} C_DIS
LIN {X -0.012,Y -553.962,Z 870.303,A 0.000,B 0.000,C 90.000,E1 270.573} C_DIS
LIN {X -0.152,Y -552.340,Z 870.303,A 0.000,B 0.000,C 90.000,E1 270.573} C_DIS
LIN {X 0.263,Y -549.841,Z 870.303,A 0.000,B 0.000,C 90.000,E1 270.458} C_DIS
LIN {X 0.233,Y -549.769,Z 870.303,A 0.000,B 0.000,C 90.000,E1 270.458} C_DIS
LIN {X 0.076,Y -546.998,Z 870.301,A 0.000,B 0.000,C 90.000,E1 270.115} C_DIS
LIN {X -0.085,Y -546.342,Z 870.299,A 0.000,B 0.000,C 90.000,E1 269.885} C_DIS
LIN {X -0.122,Y -544.890,Z 870.293,A 0.000,B 0.000,C 90.000,E1 268.797} C_DIS
LIN {X 0.211,Y -542.808,Z 870.279,A 0.000,B 0.000,C 90.000,E1 266.216} C_DIS
LIN {X -0.076,Y -541.682,Z 870.270,A 0.000,B 0.000,C 90.000,E1 264.546} C_DIS
LIN {X 0.083,Y -540.854,Z 870.263,A 0.000,B 0.000,C 90.000,E1 263.394} C_DIS
LIN {X 0.223,Y -539.920,Z 870.257,A 0.000,B 0.000,C 90.000,E1 262.243} C_DIS
LIN {X -0.047,Y -538.644,Z 870.249,A 0.000,B 0.000,C 90.000,E1 260.849} C_DIS
LIN {X 0.255,Y -536.934,Z 870.240,A 0.000,B 0.000,C 90.000,E1 259.106} C_DIS
LIN {X -0.027,Y -535.670,Z 870.233,A 0.000,B 0.000,C 90.000,E1 257.993} C_DIS
LIN {X 0.194,Y -534.396,Z 870.227,A 0.000,B 0.000,C 90.000,E1 256.825} C_DIS
LIN {X 0.217,Y -532.251,Z 870.217,A 0.000,B 0.000,C 90.000,E1 255.102} C_DIS
LIN {X 0.228,Y -529.841,Z 870.206,A 0.000,B 0.000,C 90.000,E1 253.087} C_DIS
LIN {X 0.290,Y -528.165,Z 870.198,A 0.000,B 0.000,C 90.000,E1 251.638} C_DIS
LIN {X 0.000,Y -525.897,Z 870.189,A 0.000,B 0.000,C 90.000,E1 249.934} C_DIS
LIN {X 0.170,Y -523.923,Z 870.181,A 0.000,B 0.000,C 90.000,E1 248.465} C_DIS
LIN {X -0.034,Y -521.326,Z 870.171,A 0.000,B 0.000,C 90.000,E1 246.741} C_DIS
LIN {X 0.300,Y -519.560,Z 870.164,A 0.000,B 0.000,C 90.000,E1 245.537} C_DIS
LIN {X 0.055,Y -517.303,Z 870.156,A 0.000,B 0.000,C 90.000,E1 244.101} C_DIS
LIN {X 0.098,Y -515.365,Z 870.150,A 0.000,B 0.000,C 90.000,E1 242.922} C_DIS
LIN {X 0.233,Y -512.824,Z 870.141,A 0.000,B 0.000,C 90.000,E1 241.435} C_DIS
LIN {X -0.134,Y -510.245,Z 870.133,A 0.000,B 0.000,C 90.000,E1 239.999} C_DIS
LIN {X -0.296,Y -507.560,Z 870.125,A 0.000,B 0.000,C 90.000,E1 238.535} C_DIS
LIN {X 0.071,Y -504.130,Z 870.115,A 0.000,B 0.000,C 90.000,E1 236.707} C_DIS
LIN {X 0.037,Y -501.706,Z 870.109,A 0.000,B 0.000,C 90.000,E1 235.515} C_DIS
LIN {X -0.026,Y -498.968,Z 870.102,A 0.000,B 0.000,C 90.000,E1 234.322} C_DIS
LIN {X 0.289,Y -494.620,Z 870.092,A 0.000,B 0.000,C 90.000,E1 232.477} C_DIS
LIN {X 0.101,Y -490.314,Z 870.082,A 0.000,B 0.000,C 90.000,E1 230.678} C_DIS
LIN {X 0.058,Y -486.128,Z 870.071,A 0.000,B 0.000,C 90.000,E1 228.852} C_DIS
LIN {X 0.055,Y -481.400,Z 870.060,A 0.000,B 0.000,C 90.000,E1 226.701} C_DIS
LIN {X 0.123,Y -477.358,Z 870.049,A 0.000,B 0.000,C 90.000,E1 224.838} C_DIS
LIN {X 0.008,Y -476.067,Z 870.046,A 0.000,B 0.000,C 90.000,E1 224.231} C_DIS
LIN {X 0.052,Y -471.207,Z 870.034,A 0.000,B 0.000,C 90.000,E1 222.043} C_DIS
LIN {X -0.057,Y -467.131,Z 870.023,A 0.000,B 0.000,C 90.000,E1 220.172} C_DIS
LIN {X -0.102,Y -461.705,Z 870.009,A 0.000,B 0.000,C 90.000,E1 217.649} C_DIS
LIN {X 0.277,Y -458.395,Z 870.000,A 0.000,B 0.000,C 90.000,E1 216.011} C_DIS
LIN {X 0.050,Y -454.346,Z 869.990,A 0.000,B 0.000,C 90.000,E1 214.119} C_DIS
LIN {X 0.023,Y -448.840,Z 869.975,A 0.000,B 0.000,C 90.000,E1 211.544} C_DIS
LIN {X 0.076,Y -444.635,Z 869.964,A 0.000,B 0.000,C 90.000,E1 209.589} C_DIS
LIN {X -0.073,Y -441.199,Z 869.955,A 0.000,B 0.000,C 90.000,E1 207.975} C_DIS
LIN {X -0.029,Y -436.287,Z 869.943,A 0.000,B 0.000,C 90.000,E1 205.668} C_DIS
LIN {X 0.084,Y -431.399,Z 869.930,A 0.000,B 0.000,C 90.000,E1 203.334} C_DIS
LIN {X 0.112,Y -428.031,Z 869.920,A 0.000,B 0.000,C 90.000,E1 201.663} C_DIS
LIN {X -0.141,Y -423.936,Z 869.909,A 0.000,B 0.000,C 90.000,E1 199.685} C_DIS
LIN {X -0.158,Y -420.635,Z 869.900,A 0.000,B 0.000,C 90.000,E1 198.000} C_DIS
LIN {X 0.001,Y -417.990,Z 869.892,A 0.000,B 0.000,C 90.000,E1 196.622} C_DIS
LIN {X -0.105,Y -413.818,Z 869.881,A 0.000,B 0.000,C 90.000,E1 194.592} C_DIS
LIN {X -0.006,Y -409.067,Z 869.868,A 0.000,B 0.000,C 90.000,E1 192.175} C_DIS
LIN {X 0.076,Y -406.431,Z 869.860,A 0.000,B 0.000,C 90.000,E1 190.782} C_DIS
LIN {X 0.193,Y -402.983,Z 869.850,A 0.000,B 0.000,C 90.000,E1 189.029} C_DIS
LIN {X 0.108,Y -399.461,Z 869.841,A 0.000,B 0.000,C 90.000,E1 187.296} C_DIS
LIN {X 0.092,Y -393.680,Z 869.823,A 0.000,B 0.000,C 90.000,E1 184.131} C_DIS
LIN {X -0.179,Y -388.796,Z 869.805,A 0.000,B 0.000,C 90.000,E1 180.974} C_DIS
LIN {X 0.137,Y -386.311,Z 869.795,A 0.000,B 0.000,C 90.000,E1 179.141} C_DIS
LIN {X -0.091,Y -383.212,Z 869.783,A 0.000,B 0.000,C 90.000,E1 177.020} C_DIS
LIN {X 0.157,Y -380.567,Z 869.773,A 0.000,B 0.000,C 90.000,E1 175.179} C_DIS
LIN {X -0.156,Y -374.800,Z 869.747,A 0.000,B 0.000,C 90.000,E1 170.500} C_DIS
LIN {X 0.128,Y -373.653,Z 869.739,A 0.000,B 0.000,C 90.000,E1 168.993} C_DIS
LIN {X -0.034,Y -373.386,Z 869.735,A 0.000,B 0.000,C 90.000,E1 168.285} C_DIS
LIN {X 0.171,Y -373.327,Z 869.731,A 0.000,B 0.000,C 90.000,E1 167.521} C_DIS
LIN {X -0.110,Y -373.347,Z 869.725,A 0.000,B 0.000,C 90.000,E1 166.464} C_DIS
LIN {X 0.062,Y -374.031,Z 869.719,A 0.000,B 0.000,C 90.000,E1 165.338} C_DIS
LIN {X -0.065,Y -374.421,Z 869.717,A 0.000,B 0.000,C 90.000,E1 164.991} C_DIS
LIN {X -0.094,Y -375.195,Z 869.715,A 0.000,B 0.000,C 90.000,E1 164.629} C_DIS
LIN {X -0.119,Y -375.789,Z 869.713,A 0.000,B 0.000,C 90.000,E1 164.267} C_DIS
LIN {X 0.117,Y -377.078,Z 869.711,A 0.000,B 0.000,C 90.000,E1 163.866} C_DIS
LIN {X 0.086,Y -378.979,Z 869.706,A 0.000,B 0.000,C 90.000,E1 163.142} C_DIS
LIN {X 0.077,Y -380.769,Z 869.704,A 0.000,B 0.000,C 90.000,E1 162.779} C_DIS
LIN {X 0.084,Y -384.757,Z 869.701,A 0.000,B 0.000,C 90.000,E1 162.236} C_DIS
LIN {X -0.012,Y -387.591,Z 869.700,A 0.000,B 0.000,C 90.000,E1 161.945} C_DIS
LIN {X 0.115,Y -393.115,Z 869.697,A 0.000,B 0.000,C 90.000,E1 161.511} C_DIS
LIN {X 0.002,Y -401.660,Z 869.695,A 0.000,B 0.000,C 90.000,E1 161.094} C_DIS
LIN {X -0.091,Y -408.752,Z 869.693,A 0.000,B 0.000,C 90.000,E1 160.786} C_DIS
LIN {X 0.154,Y -415.393,Z 869.691,A 0.000,B 0.000,C 90.000,E1 160.423} C_DIS
LIN {X 0.164,Y -425.334,Z 869.688,A 0.000,B 0.000,C 90.000,E1 159.880} C_DIS
LIN {X -0.057,Y -435.008,Z 869.685,A 0.000,B 0.000,C 90.000,E1 159.316} C_DIS
LIN {X -0.167,Y -444.166,Z 869.681,A 0.000,B 0.000,C 90.000,E1 158.646} C_DIS
LIN {X -0.090,Y -450.399,Z 869.679,A 0.000,B 0.000,C 90.000,E1 158.156} C_DIS
LIN {X 0.092,Y -456.277,Z 869.676,A 0.000,B 0.000,C 90.000,E1 157.614} C_DIS
LIN {X -0.162,Y -462.067,Z 869.673,A 0.000,B 0.000,C 90.000,E1 157.102} C_DIS
LIN {X -0.169,Y -467.761,Z 869.670,A 0.000,B 0.000,C 90.000,E1 156.538} C_DIS
LIN {X -0.049,Y -474.711,Z 869.666,A 0.000,B 0.000,C 90.000,E1 155.793} C_DIS
LIN {X 0.271,Y -485.061,Z 869.659,A 0.000,B 0.000,C 90.000,E1 154.588} C_DIS
LIN {X -0.104,Y -492.473,Z 869.654,A 0.000,B 0.000,C 90.000,E1 153.717} C_DIS
LIN {X -0.265,Y -497.157,Z 869.651,A 0.000,B 0.000,C 90.000,E1 153.127} C_DIS
LIN {X -0.032,Y -506.191,Z 869.644,A 0.000,B 0.000,C 90.000,E1 151.897} C_DIS
LIN {X -0.099,Y -518.776,Z 869.634,A 0.000,B 0.000,C 90.000,E1 150.127} C_DIS
LIN {X -0.045,Y -528.107,Z 869.626,A 0.000,B 0.000,C 90.000,E1 148.663} C_DIS
LIN {X 0.212,Y -530.788,Z 869.624,A 0.000,B 0.000,C 90.000,E1 148.201} C_DIS
LIN {X 0.317,Y -537.478,Z 869.617,A 0.000,B 0.000,C 90.000,E1 147.041} C_DIS
LIN {X 0.070,Y -543.854,Z 869.611,A 0.000,B 0.000,C 90.000,E1 145.928} C_DIS
LIN {X -0.136,Y -548.305,Z 869.606,A 0.000,B 0.000,C 90.000,E1 145.102} C_DIS
LIN {X -0.107,Y -553.497,Z 869.601,A 0.000,B 0.000,C 90.000,E1 144.116} C_DIS
LIN {X -0.142,Y -559.269,Z 869.594,A 0.000,B 0.000,C 90.000,E1 143.004} C_DIS
LIN {X 0.020,Y -565.618,Z 869.588,A 0.000,B 0.000,C 90.000,E1 141.743} C_DIS
LIN {X 0.183,Y -572.726,Z 869.580,A 0.000,B 0.000,C 90.000,E1 140.356} C_DIS
LIN {X 0.017,Y -575.476,Z 869.577,A 0.000,B 0.000,C 90.000,E1 139.828} C_DIS
LIN {X -0.102,Y -581.821,Z 869.569,A 0.000,B 0.000,C 90.000,E1 138.485} C_DIS
LIN {X -0.173,Y -592.843,Z 869.557,A 0.000,B 0.000,C 90.000,E1 136.215} C_DIS
LIN {X -0.046,Y -599.141,Z 869.549,A 0.000,B 0.000,C 90.000,E1 134.879} C_DIS
LIN {X 0.106,Y -605.898,Z 869.541,A 0.000,B 0.000,C 90.000,E1 133.419} C_DIS
LIN {X 0.288,Y -612.850,Z 869.533,A 0.000,B 0.000,C 90.000,E1 131.838} C_DIS
LIN {X 0.051,Y -617.281,Z 869.527,A 0.000,B 0.000,C 90.000,E1 130.825} C_DIS
LIN {X -0.062,Y -621.447,Z 869.521,A 0.000,B 0.000,C 90.000,E1 129.806} C_DIS
LIN {X 0.084,Y -627.388,Z 869.513,A 0.000,B 0.000,C 90.000,E1 128.257} C_DIS
LIN {X -0.242,Y -630.216,Z 869.508,A 0.000,B 0.000,C 90.000,E1 127.523} C_DIS
LIN {X -0.025,Y -632.222,Z 869.506,A 0.000,B 0.000,C 90.000,E1 126.996} C_DIS
LIN {X -0.315,Y -635.997,Z 869.500,A 0.000,B 0.000,C 90.000,E1 126.011} C_DIS
LIN {X -0.032,Y -639.475,Z 869.494,A 0.000,B 0.000,C 90.000,E1 124.978} C_DIS
LIN {X -0.163,Y -640.175,Z 869.493,A 0.000,B 0.000,C 90.000,E1 124.739} C_DIS
LIN {X 0.267,Y -641.914,Z 869.490,A 0.000,B 0.000,C 90.000,E1 124.199} C_DIS
LIN {X 0.157,Y -645.535,Z 869.483,A 0.000,B 0.000,C 90.000,E1 122.959} C_DIS
LIN {X -0.324,Y -646.267,Z 869.482,A 0.000,B 0.000,C 90.000,E1 122.752} C_DIS
LIN {X -0.319,Y -648.089,Z 869.478,A 0.000,B 0.000,C 90.000,E1 122.005} C_DIS
LIN {X -0.298,Y -649.772,Z 869.474,A 0.000,B 0.000,C 90.000,E1 121.258} C_DIS
LIN {X 0.297,Y -651.366,Z 869.469,A 0.000,B 0.000,C 90.000,E1 120.463} C_DIS
LIN {X -0.077,Y -652.145,Z 869.467,A 0.000,B 0.000,C 90.000,E1 120.001} C_DIS
LIN {X 0.020,Y -652.680,Z 869.465,A 0.000,B 0.000,C 90.000,E1 119.745} C_DIS
LIN {X 0.183,Y -654.268,Z 869.460,A 0.000,B 0.000,C 90.000,E1 118.743} C_DIS
LIN {X -0.067,Y -655.324,Z 869.456,A 0.000,B 0.000,C 90.000,E1 118.025} C_DIS
LIN {X 0.045,Y -655.747,Z 869.454,A 0.000,B 0.000,C 90.000,E1 117.769} C_DIS
LIN {X 0.159,Y -656.031,Z 869.453,A 0.000,B 0.000,C 90.000,E1 117.513} C_DIS
LIN {X -0.076,Y -657.240,Z 869.449,A 0.000,B 0.000,C 90.000,E1 116.796} C_DIS
LIN {X -0.004,Y -658.283,Z 869.445,A 0.000,B 0.000,C 90.000,E1 116.052} C_DIS
LIN {X 0.247,Y -658.778,Z 869.442,A 0.000,B 0.000,C 90.000,E1 115.540} C_DIS
LIN {X -0.122,Y -659.423,Z 869.437,A 0.000,B 0.000,C 90.000,E1 114.591} C_DIS
LIN {X 0.132,Y -659.637,Z 869.434,A 0.000,B 0.000,C 90.000,E1 114.079} C_DIS
LIN {X 0.118,Y -659.442,Z 869.431,A 0.000,B 0.000,C 90.000,E1 113.590} C_DIS
LIN {X 0.245,Y -659.135,Z 869.430,A 0.000,B 0.000,C 90.000,E1 113.334} C_DIS
LIN {X -0.312,Y -656.810,Z 869.426,A 0.000,B 0.000,C 90.000,E1 112.770} C_DIS
LIN {X -0.252,Y -656.030,Z 869.426,A 0.000,B 0.000,C 90.000,E1 112.642} C_DIS
LIN {X -0.282,Y -652.042,Z 869.423,A 0.000,B 0.000,C 90.000,E1 112.153} C_DIS
LIN {X -0.184,Y -648.943,Z 869.422,A 0.000,B 0.000,C 90.000,E1 111.897} C_DIS
LIN {X 0.075,Y -645.871,Z 869.420,A 0.000,B 0.000,C 90.000,E1 111.663} C_DIS
LIN {X -0.212,Y -644.218,Z 869.420,A 0.000,B 0.000,C 90.000,E1 111.589} C_DIS
LIN {X 0.099,Y -641.693,Z 869.419,A 0.000,B 0.000,C 90.000,E1 111.461} C_DIS
LIN {X 0.024,Y -635.823,Z 869.418,A 0.000,B 0.000,C 90.000,E1 111.173} C_DIS
LIN {X 0.169,Y -624.917,Z 869.415,A 0.000,B 0.000,C 90.000,E1 110.737} C_DIS
LIN {X -0.057,Y -611.760,Z 869.413,A 0.000,B 0.000,C 90.000,E1 110.248} C_DIS
LIN {X -0.182,Y -594.369,Z 869.408,A 0.000,B 0.000,C 90.000,E1 109.450} C_DIS
LIN {X -0.162,Y -587.649,Z 869.406,A 0.000,B 0.000,C 90.000,E1 109.141} C_DIS
LIN {X 0.170,Y -578.431,Z 869.404,A 0.000,B 0.000,C 90.000,E1 108.779} C_DIS
LIN {X -0.164,Y -567.625,Z 869.403,A 0.000,B 0.000,C 90.000,E1 108.489} C_DIS
LIN {X 0.058,Y -564.970,Z 869.402,A 0.000,B 0.000,C 90.000,E1 108.362} C_DIS
LIN {X 0.079,Y -562.509,Z 869.401,A 0.000,B 0.000,C 90.000,E1 108.236} C_DIS
LIN {X 0.215,Y -561.954,Z 869.401,A 0.000,B 0.000,C 90.000,E1 108.181} C_DIS
LIN {X 0.203,Y -560.485,Z 869.400,A 0.000,B 0.000,C 90.000,E1 108.000} C_DIS
LIN {X 0.089,Y -559.918,Z 869.399,A 0.000,B 0.000,C 90.000,E1 107.873} C_DIS
LIN {X 0.221,Y -558.999,Z 869.398,A 0.000,B 0.000,C 90.000,E1 107.583} C_DIS
LIN {X -0.299,Y -558.547,Z 869.396,A 0.000,B 0.000,C 90.000,E1 107.221} C_DIS
LIN {X -0.079,Y -559.334,Z 869.375,A 0.000,B 0.000,C 90.000,E1 103.592} C_DIS
LIN {X -0.292,Y -560.212,Z 869.366,A 0.000,B 0.000,C 90.000,E1 101.951} C_DIS
LIN {X 0.064,Y -561.349,Z 869.357,A 0.000,B 0.000,C 90.000,E1 100.254} C_DIS
LIN {X 0.029,Y -562.149,Z 869.351,A 0.000,B 0.000,C 90.000,E1 99.151} C_DIS
LIN {X 0.241,Y -563.294,Z 869.342,A 0.000,B 0.000,C 90.000,E1 97.473} C_DIS
LIN {X 0.228,Y -563.969,Z 869.336,A 0.000,B 0.000,C 90.000,E1 96.372} C_DIS
LIN {X -0.163,Y -564.757,Z 869.326,A 0.000,B 0.000,C 90.000,E1 94.759} C_DIS
LIN {X -0.028,Y -565.391,Z 869.317,A 0.000,B 0.000,C 90.000,E1 93.094} C_DIS
LIN {X 0.205,Y -566.008,Z 869.307,A 0.000,B 0.000,C 90.000,E1 91.146} C_DIS
LIN {X -0.234,Y -566.430,Z 869.297,A 0.000,B 0.000,C 90.000,E1 89.542} C_DIS
LIN {X -0.203,Y -566.673,Z 869.290,A 0.000,B 0.000,C 90.000,E1 88.165} C_DIS
LIN {X -0.046,Y -566.959,Z 869.281,A 0.000,B 0.000,C 90.000,E1 86.502} C_DIS
LIN {X 0.143,Y -567.274,Z 869.271,A 0.000,B 0.000,C 90.000,E1 84.837} C_DIS
LIN {X -0.178,Y -567.571,Z 869.262,A 0.000,B 0.000,C 90.000,E1 83.223} C_DIS
LIN {X 0.022,Y -568.234,Z 869.249,A 0.000,B 0.000,C 90.000,E1 80.735} C_DIS
LIN {X 0.261,Y -568.708,Z 869.241,A 0.000,B 0.000,C 90.000,E1 79.342} C_DIS
LIN {X 0.051,Y -569.678,Z 869.229,A 0.000,B 0.000,C 90.000,E1 77.173} C_DIS
LIN {X -0.002,Y -570.146,Z 869.221,A 0.000,B 0.000,C 90.000,E1 75.811} C_DIS
LIN {X 0.140,Y -570.718,Z 869.212,A 0.000,B 0.000,C 90.000,E1 74.157} C_DIS
LIN {X 0.262,Y -571.029,Z 869.205,A 0.000,B 0.000,C 90.000,E1 72.779} C_DIS
LIN {X 0.194,Y -571.241,Z 869.195,A 0.000,B 0.000,C 90.000,E1 71.148} C_DIS
LIN {X -0.057,Y -571.395,Z 869.185,A 0.000,B 0.000,C 90.000,E1 69.263} C_DIS
LIN {X -0.112,Y -571.402,Z 869.174,A 0.000,B 0.000,C 90.000,E1 67.358} C_DIS
LIN {X 0.090,Y -571.422,Z 869.167,A 0.000,B 0.000,C 90.000,E1 65.973} C_DIS
LIN {X 0.296,Y -571.278,Z 869.159,A 0.000,B 0.000,C 90.000,E1 64.588} C_DIS
LIN {X -0.022,Y -571.017,Z 869.151,A 0.000,B 0.000,C 90.000,E1 63.256} C_DIS
LIN {X -0.259,Y -570.556,Z 869.142,A 0.000,B 0.000,C 90.000,E1 61.641} C_DIS
LIN {X -0.170,Y -570.149,Z 869.136,A 0.000,B 0.000,C 90.000,E1 60.539} C_DIS
LIN {X -0.124,Y -569.813,Z 869.132,A 0.000,B 0.000,C 90.000,E1 59.715} C_DIS
LIN {X -0.125,Y -568.623,Z 869.123,A 0.000,B 0.000,C 90.000,E1 58.074} C_DIS
LIN {X -0.081,Y -567.978,Z 869.118,A 0.000,B 0.000,C 90.000,E1 57.248} C_DIS
LIN {X -0.157,Y -567.503,Z 869.115,A 0.000,B 0.000,C 90.000,E1 56.707} C_DIS
LIN {X -0.008,Y -566.245,Z 869.109,A 0.000,B 0.000,C 90.000,E1 55.595} C_DIS
LIN {X 0.125,Y -564.816,Z 869.103,A 0.000,B 0.000,C 90.000,E1 54.482} C_DIS
LIN {X -0.224,Y -563.203,Z 869.097,A 0.000,B 0.000,C 90.000,E1 53.417} C_DIS
LIN {X 0.090,Y -561.857,Z 869.092,A 0.000,B 0.000,C 90.000,E1 52.557} C_DIS
LIN {X -0.054,Y -560.344,Z 869.087,A 0.000,B 0.000,C 90.000,E1 51.743} C_DIS
LIN {X 0.225,Y -558.640,Z 869.083,A 0.000,B 0.000,C 90.000,E1 50.884} C_DIS
LIN {X 0.047,Y -556.631,Z 869.078,A 0.000,B 0.000,C 90.000,E1 50.070} C_DIS
LIN {X 0.209,Y -554.296,Z 869.074,A 0.000,B 0.000,C 90.000,E1 49.218} C_DIS
LIN {X -0.075,Y -552.651,Z 869.070,A 0.000,B 0.000,C 90.000,E1 48.690} C_DIS
LIN {X 0.049,Y -549.781,Z 869.066,A 0.000,B 0.000,C 90.000,E1 47.838} C_DIS
LIN {X 0.143,Y -546.553,Z 869.061,A 0.000,B 0.000,C 90.000,E1 46.986} C_DIS
